(* IEC 61131-3 sources: cc_kush_rewrite/POUs (part 3) *)

FC_ModbusWriteBool(pRegisters := ADR(awModbusInputRegisters), iRegisterIndex := 355, iBitIndex := 0, xValue := stBunker[2].MotorVibrator[3].qxKM_Power);
FC_ModbusWriteBool(pRegisters := ADR(awModbusInputRegisters), iRegisterIndex := 355, iBitIndex := 1, xValue := stBunker[2].MotorVibrator[4].qxKM_Power);
FC_ModbusWriteBool(pRegisters := ADR(awModbusInputRegisters), iRegisterIndex := 355, iBitIndex := 2, xValue := stBunker[3].MotorVibFeeder[1].qxKM_Power);
FC_ModbusWriteBool(pRegisters := ADR(awModbusInputRegisters), iRegisterIndex := 355, iBitIndex := 3, xValue := stBunker[3].MotorVibFeeder[2].qxKM_Power);
FC_ModbusWriteBool(pRegisters := ADR(awModbusInputRegisters), iRegisterIndex := 355, iBitIndex := 4, xValue := stBunker[3].MotorVibrator[1].qxKM_Power);
FC_ModbusWriteBool(pRegisters := ADR(awModbusInputRegisters), iRegisterIndex := 355, iBitIndex := 5, xValue := stBunker[3].MotorVibrator[2].qxKM_Power);
FC_ModbusWriteBool(pRegisters := ADR(awModbusInputRegisters), iRegisterIndex := 355, iBitIndex := 6, xValue := stBunker[3].MotorVibrator[3].qxKM_Power);
FC_ModbusWriteBool(pRegisters := ADR(awModbusInputRegisters), iRegisterIndex := 355, iBitIndex := 7, xValue := stBunker[3].MotorVibrator[4].qxKM_Power);
FC_ModbusWriteBool(pRegisters := ADR(awModbusInputRegisters), iRegisterIndex := 355, iBitIndex := 8, xValue := stConveyor.xHLA);
FC_ModbusWriteBool(pRegisters := ADR(awModbusInputRegisters), iRegisterIndex := 355, iBitIndex := 10, xValue := stDumper.xHLA);
FC_ModbusWriteBool(pRegisters := ADR(awModbusInputRegisters), iRegisterIndex := 355, iBitIndex := 11, xValue := stCommonSignals.qx6KM1);
FC_ModbusWriteBool(pRegisters := ADR(awModbusInputRegisters), iRegisterIndex := 355, iBitIndex := 12, xValue := stConveyor.qxBreakerConveyor);
FC_ModbusWriteBool(pRegisters := ADR(awModbusInputRegisters), iRegisterIndex := 355, iBitIndex := 13, xValue := stDumper.qxBreakerConveyor);
FC_ModbusWriteBool(pRegisters := ADR(awModbusInputRegisters), iRegisterIndex := 355, iBitIndex := 14, xValue := stDumper.qxBreakerRotation);

// Модуль DO4 (356-357): Светофоры бункеров
FC_ModbusWriteBool(pRegisters := ADR(awModbusInputRegisters), iRegisterIndex := 356, iBitIndex := 0, xValue := stBunker[1].qxLightRed);
FC_ModbusWriteBool(pRegisters := ADR(awModbusInputRegisters), iRegisterIndex := 356, iBitIndex := 1, xValue := stBunker[1].qxLightYellow);
FC_ModbusWriteBool(pRegisters := ADR(awModbusInputRegisters), iRegisterIndex := 356, iBitIndex := 2, xValue := stBunker[1].qxLightGreen);
FC_ModbusWriteBool(pRegisters := ADR(awModbusInputRegisters), iRegisterIndex := 356, iBitIndex := 3, xValue := stBunker[2].qxLightRed);
FC_ModbusWriteBool(pRegisters := ADR(awModbusInputRegisters), iRegisterIndex := 356, iBitIndex := 4, xValue := stBunker[2].qxLightYellow);
FC_ModbusWriteBool(pRegisters := ADR(awModbusInputRegisters), iRegisterIndex := 356, iBitIndex := 5, xValue := stBunker[2].qxLightGreen);
FC_ModbusWriteBool(pRegisters := ADR(awModbusInputRegisters), iRegisterIndex := 356, iBitIndex := 6, xValue := stBunker[3].qxLightRed);
FC_ModbusWriteBool(pRegisters := ADR(awModbusInputRegisters), iRegisterIndex := 356, iBitIndex := 7, xValue := stBunker[3].qxLightYellow);
FC_ModbusWriteBool(pRegisters := ADR(awModbusInputRegisters), iRegisterIndex := 356, iBitIndex := 8, xValue := stBunker[3].qxLightGreen);

END_FUNCTION_BLOCK

(* ---- FB_Simulation.st ---- *)
FUNCTION_BLOCK FB_Simulation
VAR_INPUT
	xEnable : BOOL; // Включение симуляции
	xReset : BOOL; // Сброс всех переменных (симуляция отсутствия ошибок)
	Dumper : REFERENCE TO ST_Dumper; // Структура отвалообразователя
	Conveyor : REFERENCE TO ST_ConveyorPrefabricated; // Структура сборного конвейера
	Bunker : REFERENCE TO ARRAY[1..3] OF ST_Bunker; // Массив бункеров
	Common : ST_CommonSignals; // Общие сигналы
	tFeedbackDelay : TIME := T#500MS; // Задержка обратной связи
END_VAR
VAR
	// Детекция переднего фронта
	rtEnable : R_TRIG;
	rtReset : R_TRIG;

	// Флаг инициализации
	_xInitRequired : BOOL;

	// Индексы для циклов
	b, m : INT;

	// === Симуляция веса бункеров ===
	// Средняя частота вибропитателей каждого бункера
	_rAvgFrequencyVibFeeder : ARRAY[1..3] OF REAL;

	// Скорость расхода веса бункера (кг/с) в зависимости от частоты вибропитателей
	_rWeightDischargeRate : ARRAY[1..3] OF REAL;

	// Скорость заполнения веса бункера (кг/с) в зависимости от светофора
	_rWeightFillRate : ARRAY[1..3] OF REAL;

	// Таймер для периодического заполнения по приоритету
	_tonFillTimer : ARRAY[1..3] OF TON;
	_xFillTimerActive : ARRAY[1..3] OF BOOL;

	// Параметры заполнения (настраиваются через входные параметры)
	_rFillRateGreen : REAL := 0.8; // Скорость заполнения на зелёном (кг/с) - плавное заполнение
	_rFillRateYellow : REAL := 0.3; // Скорость заполнения на жёлтом (кг/с) - медленное заполнение
	_tFillPeriod : TIME := T#8S; // Период заполнения (раз в N секунд) - реже
	_tFillDuration : TIME := T#3S; // Длительность одного заполнения - дольше

	// Константа расхода: частота 50 Гц → 0.5 кг/с расход (замедлено)
	_rDischargeCoeff : REAL := 0.01; // 50 Гц * 0.01 = 0.5 кг/с

	// === Симуляция веса под бункерами ===

	// Скорость накопления веса (кг/с) для каждого бункера
	_rWeightAccumulationRate : ARRAY[1..3] OF REAL;

	// Накопленный вес от каждого бункера (независимо)
	_rLocalWeightUnderBunker : ARRAY[1..3] OF REAL;

	// === Случайные возмущения для бункеров ===
	// Параметры генератора псевдослучайных чисел (Linear Congruential Generator)
	_nRandomSeed : ARRAY[1..3] OF DINT := [12345, 67890, 24680]; // Начальные значения

	// Случайное смещение для каждого бункера (-1.0 до +1.0)
	_rRandomOffset : ARRAY[1..3] OF REAL;

	// Линейный дрейф (медленное изменение характеристик материала)
	_rDriftOffset : ARRAY[1..3] OF REAL;
	_rDriftSpeed : ARRAY[1..3] OF REAL := [0.0003, -0.00025, 0.00035]; // Скорость дрейфа за цикл

	// Временные переменные
	_rNoise : REAL; // Шум ±3%
	_rDrift : REAL; // Дрейф ±8%

	// === Таймеры отвалообразователя ===
	// Таймеры обратной связи контакторов (KM)
	tonKM_Conv1, tonKM_Conv2 : TON;
	tonKM_Rot1, tonKM_Rot2 : TON;

	// Таймеры обратной связи ЧРП (IsWorking)
	tonVFD_Conv1, tonVFD_Conv2 : TON;
	tonVFD_Rot1, tonVFD_Rot2 : TON;

	// Таймеры обратной связи тормозов отвалообразователя
	tonBreaker_DumperConv, tonBreaker_DumperRot : TON;

	// === Таймеры сборного конвейера ===
	// Таймеры обратной связи контакторов (KM)
	tonKM_PrefConv1, tonKM_PrefConv2 : TON;

	// Таймеры обратной связи ЧРП (IsWorking)
	tonVFD_PrefConv1, tonVFD_PrefConv2 : TON;

	// Таймер обратной связи тормоза сборного конвейера
	tonBreaker_PrefConv : TON;

	// === Таймеры бункеров ===
	// Таймеры обратной связи вибропитателей [бункер 1..3][мотор 1..2]
	tonKM_VibFeeder : ARRAY[1..3, 1..2] OF TON;
	tonVFD_VibFeeder : ARRAY[1..3, 1..2] OF TON;

	// Таймеры обратной связи вибраторов [бункер 1..3][мотор 1..4]
	tonKM_Vibrator : ARRAY[1..3, 1..4] OF TON;
	tonVFD_Vibrator : ARRAY[1..3, 1..4] OF TON;

	// ========================================
	// ПЕРЕМЕННЫЕ ДЛЯ ОТЛАДКИ - СИМУЛЯЦИЯ ОБРАТНОЙ СВЯЗИ VFD
	// TRUE = обратная связь есть (нормальная работа)
	// FALSE = обратная связь отсутствует (ошибка - нет обратной связи)
	// ========================================

	// Отвалообразователь - моторы конвейера
	_xSimVFDFeedback_DumperConv1 : BOOL := TRUE;
	_xSimVFDFeedback_DumperConv2 : BOOL := TRUE;

	// Отвалообразователь - моторы поворота
	_xSimVFDFeedback_DumperRot1 : BOOL := TRUE;
	_xSimVFDFeedback_DumperRot2 : BOOL := TRUE;

	// Сборный конвейер - моторы конвейера
	_xSimVFDFeedback_ConveyorConv1 : BOOL := TRUE;
	_xSimVFDFeedback_ConveyorConv2 : BOOL := TRUE;

	// Бункеры - вибропитатели [бункер 1..3][мотор 1..2]
	_xSimVFDFeedback_VibFeeder : ARRAY[1..3, 1..2] OF BOOL := [TRUE, TRUE, TRUE, TRUE, TRUE, TRUE];

	// Бункеры - вибраторы [бункер 1..3][мотор 1..4]
	_xSimVFDFeedback_Vibrator : ARRAY[1..3, 1..4] OF BOOL := [
		TRUE, TRUE, TRUE, TRUE,
		TRUE, TRUE, TRUE, TRUE,
		TRUE, TRUE, TRUE, TRUE
	];
END_VAR

// Детекция фронтов
rtEnable(CLK := xEnable);
rtReset(CLK := xReset);

// Инициализация по переднему фронту Enable или Reset
_xInitRequired := rtEnable.Q OR rtReset.Q;

IF _xInitRequired THEN

	// ========================================
	// ИНИЦИАЛИЗАЦИЯ ОБЩИЕ СИГНАЛЫ
	// ========================================

	// Кнопка аварийной остановки - инвертированный сигнал (NC)
	Common.fbEmergencyStopBtn.ixSignal := TRUE;

	// Сигнал ПМУ - режим управления 1 - дистанция, 0 - местный
	Common.fbRemoteModeBtn.ixSignal := TRUE;

	// ========================================
	// ИНИЦИАЛИЗАЦИЯ СИМУЛЯЦИИ ОТВАЛООБРАЗОВАТЕЛЯ
	// Установка всех сигналов в состояние "нет ошибок"
	// ========================================

	// Моторы конвейера - ЧРП готовность
	Dumper.MotorConveyor[1].VFD.fbStateRdyToStart.ixSignal := TRUE;
	Dumper.MotorConveyor[2].VFD.fbStateRdyToStart.ixSignal := TRUE;

	// Моторы поворота - ЧРП готовность
	Dumper.MotorRotation[1].VFD.fbStateRdyToStart.ixSignal := TRUE;
	Dumper.MotorRotation[2].VFD.fbStateRdyToStart.ixSignal := TRUE;

	// Автоматические выключатели (QF)
	Dumper.MotorConveyor[1].fbStateQF.ixSignal := TRUE;
	Dumper.MotorConveyor[2].fbStateQF.ixSignal := TRUE;
	Dumper.MotorRotation[1].fbStateQF.ixSignal := TRUE;
	Dumper.MotorRotation[2].fbStateQF.ixSignal := TRUE;

	// ЧРП ошибки - инвертированный сигнал (NC)
	Dumper.MotorConveyor[1].VFD.fbStateFailure.ixSignal := TRUE;
	Dumper.MotorConveyor[2].VFD.fbStateFailure.ixSignal := TRUE;
	Dumper.MotorRotation[1].VFD.fbStateFailure.ixSignal := TRUE;
	Dumper.MotorRotation[2].VFD.fbStateFailure.ixSignal := TRUE;

	// Перегрев статора - инвертированный сигнал (NC)
	Dumper.MotorConveyor[1].fbStatorOverheat.ixSignal := TRUE;
	Dumper.MotorConveyor[2].fbStatorOverheat.ixSignal := TRUE;
	Dumper.MotorRotation[1].fbStatorOverheat.ixSignal := TRUE;
	Dumper.MotorRotation[2].fbStatorOverheat.ixSignal := TRUE;

	// Кабель-тросовые выключатели (HQ)
	Dumper.fbHQ_IsOk[1].ixSignal := TRUE;
	Dumper.fbHQ_IsOk[2].ixSignal := TRUE;
	Dumper.fbHQ_IsOk[3].ixSignal := TRUE;
	Dumper.fbHQ_IsOk[4].ixSignal := TRUE;

	// Контроль ограждения барабана (SQ)
	Dumper.fbSQ_IsOk[1].ixSignal := TRUE;
	Dumper.fbSQ_IsOk[2].ixSignal := TRUE;

	// Контроль схода ленты - тревога (ZQ) - инвертированный сигнал (NC)
	Dumper.fbZQAlarm[1].ixSignal := TRUE;
	Dumper.fbZQAlarm[2].ixSignal := TRUE;
	Dumper.fbZQAlarm[3].ixSignal := TRUE;
	Dumper.fbZQAlarm[4].ixSignal := TRUE;

	// Контроль схода ленты - предупреждение (ZQ) - инвертированный сигнал (NC)
	Dumper.fbZQWarning[1].ixSignal := TRUE;
	Dumper.fbZQWarning[2].ixSignal := TRUE;
	Dumper.fbZQWarning[3].ixSignal := TRUE;
	Dumper.fbZQWarning[4].ixSignal := TRUE;

	// Кнопка аварийной остановки - инвертированный сигнал (NC)
	Dumper.fbBtnEmergencyStop.ixSignal := TRUE;

	// Концевые выключатели - инвертированный сигнал (NC)
	Dumper.fbEndSwitchLeft.ixSignal := TRUE;
	Dumper.fbEndSwitchRight.ixSignal := TRUE;

	// Контроль заштыбовки - норма = 1
	Dumper.fbGS1.ixSignal := TRUE;

	// Контроль продольного разрыва ленты - норма = 1
	Dumper.fbYS1.ixSignal := TRUE;

	// Тормоза - в начале активны (NOT released)
	Dumper.fbBreakerConveyor.ixSignal := FALSE;
	Dumper.fbBreakerRotation.ixSignal := FALSE;

	// ========================================
	// ИНИЦИАЛИЗАЦИЯ СИМУЛЯЦИИ СБОРНОГО КОНВЕЙЕРА
	// Установка всех сигналов в состояние "нет ошибок"
	// ========================================

	// Моторы конвейера - ЧРП готовность
	Conveyor.MotorConveyor[1].VFD.fbStateRdyToStart.ixSignal := TRUE;
	Conveyor.MotorConveyor[2].VFD.fbStateRdyToStart.ixSignal := TRUE;

	// Автоматические выключатели (QF)
	Conveyor.MotorConveyor[1].fbStateQF.ixSignal := TRUE;
	Conveyor.MotorConveyor[2].fbStateQF.ixSignal := TRUE;

	// ЧРП ошибки - инвертированный сигнал (NC)
	Conveyor.MotorConveyor[1].VFD.fbStateFailure.ixSignal := TRUE;
	Conveyor.MotorConveyor[2].VFD.fbStateFailure.ixSignal := TRUE;

	// Перегрев статора - инвертированный сигнал (NC)
	Conveyor.MotorConveyor[1].fbStatorOverheat.ixSignal := TRUE;
	Conveyor.MotorConveyor[2].fbStatorOverheat.ixSignal := TRUE;

	// Кабель-тросовые выключатели (HQ)
	Conveyor.fbHQ_IsOk[1].ixSignal := TRUE;
	Conveyor.fbHQ_IsOk[2].ixSignal := TRUE;
	Conveyor.fbHQ_IsOk[3].ixSignal := TRUE;
	Conveyor.fbHQ_IsOk[4].ixSignal := TRUE;

	// Контроль ограждения барабана (SQ)
	Conveyor.fbSQ_IsOk[1].ixSignal := TRUE;
	Conveyor.fbSQ_IsOk[2].ixSignal := TRUE;

	// Контроль схода ленты - тревога (ZQ) - инвертированный сигнал (NC)
	Conveyor.fbZQAlarm[1].ixSignal := TRUE;
	Conveyor.fbZQAlarm[2].ixSignal := TRUE;
	Conveyor.fbZQAlarm[3].ixSignal := TRUE;
	Conveyor.fbZQAlarm[4].ixSignal := TRUE;

	// Контроль схода ленты - предупреждение (ZQ) - инвертированный сигнал (NC)
	Conveyor.fbZQWarning[1].ixSignal := TRUE;
	Conveyor.fbZQWarning[2].ixSignal := TRUE;
	Conveyor.fbZQWarning[3].ixSignal := TRUE;
	Conveyor.fbZQWarning[4].ixSignal := TRUE;

	// Кнопка аварийной остановки - инвертированный сигнал (NC)
	Conveyor.fbBtnEmergencyStop.ixSignal := TRUE;

	// Контроль заштыбовки - норма = 1
	Conveyor.fbGS1.ixSignal := TRUE;

	// Контроль продольного разрыва ленты - норма = 1
	Conveyor.fbYS1.ixSignal := TRUE;

	// Металлодетектор - норма = 0 (металл не обнаружен)
	Conveyor.fbYE1.ixSignal := FALSE;

	// ========================================
	// ИНИЦИАЛИЗАЦИЯ СИМУЛЯЦИИ БУНКЕРОВ
	// Установка всех сигналов в состояние "нет ошибок"
	// ========================================

	// ========================================
	// БУНКЕР 1
	// ========================================

	// Вибропитатели (MotorVibFeeder[1..2])
	// Вибропитатель 1
	Bunker[1].MotorVibFeeder[1].VFD.fbStateRdyToStart.ixSignal := TRUE;
	Bunker[1].MotorVibFeeder[1].fbStateQF.ixSignal := TRUE;
	Bunker[1].MotorVibFeeder[1].VFD.fbStateFailure.ixSignal := TRUE;
	Bunker[1].MotorVibFeeder[1].fbStatorOverheat.ixSignal := TRUE;

	// Вибропитатель 2
	Bunker[1].MotorVibFeeder[2].VFD.fbStateRdyToStart.ixSignal := TRUE;
	Bunker[1].MotorVibFeeder[2].fbStateQF.ixSignal := TRUE;
	Bunker[1].MotorVibFeeder[2].VFD.fbStateFailure.ixSignal := TRUE;
	Bunker[1].MotorVibFeeder[2].fbStatorOverheat.ixSignal := TRUE;

	// Вибраторы (MotorVibrator[1..4])
	Bunker[1].MotorVibrator[1].VFD.fbStateRdyToStart.ixSignal := TRUE;
	Bunker[1].MotorVibrator[1].fbStateQF.ixSignal := TRUE;
	Bunker[1].MotorVibrator[1].VFD.fbStateFailure.ixSignal := TRUE;

	Bunker[1].MotorVibrator[2].VFD.fbStateRdyToStart.ixSignal := TRUE;
	Bunker[1].MotorVibrator[2].fbStateQF.ixSignal := TRUE;
	Bunker[1].MotorVibrator[2].VFD.fbStateFailure.ixSignal := TRUE;

	Bunker[1].MotorVibrator[3].VFD.fbStateRdyToStart.ixSignal := TRUE;
	Bunker[1].MotorVibrator[3].fbStateQF.ixSignal := TRUE;
	Bunker[1].MotorVibrator[3].VFD.fbStateFailure.ixSignal := TRUE;

	Bunker[1].MotorVibrator[4].VFD.fbStateRdyToStart.ixSignal := TRUE;
	Bunker[1].MotorVibrator[4].fbStateQF.ixSignal := TRUE;
	Bunker[1].MotorVibrator[4].VFD.fbStateFailure.ixSignal := TRUE;

	// Люк бункера - закрыт (норма = 1)
	Bunker[1].fbStateHatch.ixSignal := TRUE;

	// Кнопка аварийной остановки - инвертированный сигнал (NC)
	Bunker[1].fbBtnEmergencyStop.ixSignal := TRUE;

	// Начальный вес бункера (симуляция заполненного бункера)
	Bunker[1].rWeight := 100.0;

	// Сброс веса под бункером
	Bunker[1].rWeightUnderBunker := 0.0;
	_rLocalWeightUnderBunker[1] := 0.0;

	// Сброс дрейфа
	_rDriftOffset[1] := 0.0;

	// ========================================
	// БУНКЕР 2
	// ========================================

	// Вибропитатели (MotorVibFeeder[1..2])
	// Вибропитатель 1
	Bunker[2].MotorVibFeeder[1].VFD.fbStateRdyToStart.ixSignal := TRUE;
	Bunker[2].MotorVibFeeder[1].fbStateQF.ixSignal := TRUE;
	Bunker[2].MotorVibFeeder[1].VFD.fbStateFailure.ixSignal := TRUE;
	Bunker[2].MotorVibFeeder[1].fbStatorOverheat.ixSignal := TRUE;

	// Вибропитатель 2
	Bunker[2].MotorVibFeeder[2].VFD.fbStateRdyToStart.ixSignal := TRUE;
	Bunker[2].MotorVibFeeder[2].fbStateQF.ixSignal := TRUE;
	Bunker[2].MotorVibFeeder[2].VFD.fbStateFailure.ixSignal := TRUE;
	Bunker[2].MotorVibFeeder[2].fbStatorOverheat.ixSignal := TRUE;

	// Вибраторы (MotorVibrator[1..4])
	Bunker[2].MotorVibrator[1].VFD.fbStateRdyToStart.ixSignal := TRUE;
	Bunker[2].MotorVibrator[1].fbStateQF.ixSignal := TRUE;
	Bunker[2].MotorVibrator[1].VFD.fbStateFailure.ixSignal := TRUE;

	Bunker[2].MotorVibrator[2].VFD.fbStateRdyToStart.ixSignal := TRUE;
	Bunker[2].MotorVibrator[2].fbStateQF.ixSignal := TRUE;
	Bunker[2].MotorVibrator[2].VFD.fbStateFailure.ixSignal := TRUE;

	Bunker[2].MotorVibrator[3].VFD.fbStateRdyToStart.ixSignal := TRUE;
	Bunker[2].MotorVibrator[3].fbStateQF.ixSignal := TRUE;
	Bunker[2].MotorVibrator[3].VFD.fbStateFailure.ixSignal := TRUE;

	Bunker[2].MotorVibrator[4].VFD.fbStateRdyToStart.ixSignal := TRUE;
	Bunker[2].MotorVibrator[4].fbStateQF.ixSignal := TRUE;
	Bunker[2].MotorVibrator[4].VFD.fbStateFailure.ixSignal := TRUE;

	// Люк бункера - закрыт (норма = 1)
	Bunker[2].fbStateHatch.ixSignal := TRUE;

	// Кнопка аварийной остановки - инвертированный сигнал (NC)
	Bunker[2].fbBtnEmergencyStop.ixSignal := TRUE;

	// Начальный вес бункера (симуляция заполненного бункера)
	Bunker[2].rWeight := 100.0;

	// Сброс веса под бункером
	Bunker[2].rWeightUnderBunker := 0.0;
	_rLocalWeightUnderBunker[2] := 0.0;

	// Сброс дрейфа
	_rDriftOffset[2] := 0.0;

	// ========================================
	// БУНКЕР 3
	// ========================================

	// Вибропитатели (MotorVibFeeder[1..2])
	// Вибропитатель 1
	Bunker[3].MotorVibFeeder[1].VFD.fbStateRdyToStart.ixSignal := TRUE;
	Bunker[3].MotorVibFeeder[1].fbStateQF.ixSignal := TRUE;
	Bunker[3].MotorVibFeeder[1].VFD.fbStateFailure.ixSignal := TRUE;
	Bunker[3].MotorVibFeeder[1].fbStatorOverheat.ixSignal := TRUE;

	// Вибропитатель 2
	Bunker[3].MotorVibFeeder[2].VFD.fbStateRdyToStart.ixSignal := TRUE;
	Bunker[3].MotorVibFeeder[2].fbStateQF.ixSignal := TRUE;
	Bunker[3].MotorVibFeeder[2].VFD.fbStateFailure.ixSignal := TRUE;
	Bunker[3].MotorVibFeeder[2].fbStatorOverheat.ixSignal := TRUE;

	// Вибраторы (MotorVibrator[1..4])
	Bunker[3].MotorVibrator[1].VFD.fbStateRdyToStart.ixSignal := TRUE;
	Bunker[3].MotorVibrator[1].fbStateQF.ixSignal := TRUE;
	Bunker[3].MotorVibrator[1].VFD.fbStateFailure.ixSignal := TRUE;

	Bunker[3].MotorVibrator[2].VFD.fbStateRdyToStart.ixSignal := TRUE;
	Bunker[3].MotorVibrator[2].fbStateQF.ixSignal := TRUE;
	Bunker[3].MotorVibrator[2].VFD.fbStateFailure.ixSignal := TRUE;

	Bunker[3].MotorVibrator[3].VFD.fbStateRdyToStart.ixSignal := TRUE;
	Bunker[3].MotorVibrator[3].fbStateQF.ixSignal := TRUE;
	Bunker[3].MotorVibrator[3].VFD.fbStateFailure.ixSignal := TRUE;

	Bunker[3].MotorVibrator[4].VFD.fbStateRdyToStart.ixSignal := TRUE;
	Bunker[3].MotorVibrator[4].fbStateQF.ixSignal := TRUE;
	Bunker[3].MotorVibrator[4].VFD.fbStateFailure.ixSignal := TRUE;

	// Люк бункера - закрыт (норма = 1)
	Bunker[3].fbStateHatch.ixSignal := TRUE;

	// Кнопка аварийной остановки - инвертированный сигнал (NC)
	Bunker[3].fbBtnEmergencyStop.ixSignal := TRUE;

	// Начальный вес бункера (симуляция заполненного бункера)
	Bunker[3].rWeight := 100.0;

	// Сброс веса под бункером
	Bunker[3].rWeightUnderBunker := 0.0;
	_rLocalWeightUnderBunker[3] := 0.0;

	// Сброс дрейфа
	_rDriftOffset[3] := 0.0;
END_IF;

// ========================================
// ПРОЦЕСС СИМУЛЯЦИИ
// ========================================

IF xEnable THEN
	// ========================================
	// СИМУЛЯЦИЯ ОТВАЛООБРАЗОВАТЕЛЯ
	// ========================================

	// Симуляция частоты ЧРП моторов конвейера отвалообразователя
	// В режиме симуляции FB_AnalogInput использует refSimValue (rSimulatedFrequency) напрямую,
	// поэтому записываем целевую частоту в rSimulatedFrequency
	Dumper.MotorConveyor[1].VFD.rSimulatedFrequency := Dumper.MotorConveyor[1].VFD.qrOutFrequency;
	Dumper.MotorConveyor[2].VFD.rSimulatedFrequency := Dumper.MotorConveyor[2].VFD.qrOutFrequency;

	// Симуляция частоты ЧРП моторов поворота отвалообразователя
	Dumper.MotorRotation[1].VFD.rSimulatedFrequency := Dumper.MotorRotation[1].VFD.qrOutFrequency;
	Dumper.MotorRotation[2].VFD.rSimulatedFrequency := Dumper.MotorRotation[2].VFD.qrOutFrequency;

	// ========================================
	// СИМУЛЯЦИЯ ОБРАТНОЙ СВЯЗИ ОТВАЛООБРАЗОВАТЕЛЯ
	// ========================================

	// Обратная связь контакторов моторов конвейера отвалообразователя
	tonKM_Conv1(IN := Dumper.MotorConveyor[1].qxKM_Power, PT := tFeedbackDelay);
	Dumper.MotorConveyor[1].fbStateKM.ixSignal := tonKM_Conv1.Q;

	tonKM_Conv2(IN := Dumper.MotorConveyor[2].qxKM_Power, PT := tFeedbackDelay);
	Dumper.MotorConveyor[2].fbStateKM.ixSignal := tonKM_Conv2.Q;

	// Обратная связь контакторов моторов поворота отвалообразователя
	tonKM_Rot1(IN := Dumper.MotorRotation[1].qxKM_Power, PT := tFeedbackDelay);
	Dumper.MotorRotation[1].fbStateKM.ixSignal := tonKM_Rot1.Q;

	tonKM_Rot2(IN := Dumper.MotorRotation[2].qxKM_Power, PT := tFeedbackDelay);
	Dumper.MotorRotation[2].fbStateKM.ixSignal := tonKM_Rot2.Q;

	// Обратная связь работы ЧРП моторов конвейера отвалообразователя
	tonVFD_Conv1(IN := Dumper.MotorConveyor[1].VFD.qxStart, PT := tFeedbackDelay);
	Dumper.MotorConveyor[1].VFD.fbStateIsWorking.ixSignal := tonVFD_Conv1.Q AND _xSimVFDFeedback_DumperConv1;

	tonVFD_Conv2(IN := Dumper.MotorConveyor[2].VFD.qxStart, PT := tFeedbackDelay);
	Dumper.MotorConveyor[2].VFD.fbStateIsWorking.ixSignal := tonVFD_Conv2.Q AND _xSimVFDFeedback_DumperConv2;

	// Обратная связь работы ЧРП моторов поворота отвалообразователя
	// Учитываем как прямое, так и реверсивное вращение
	tonVFD_Rot1(IN := (Dumper.MotorRotation[1].VFD.qxStart OR Dumper.MotorRotation[1].qxVFDReverseStart), PT := tFeedbackDelay);
	Dumper.MotorRotation[1].VFD.fbStateIsWorking.ixSignal := tonVFD_Rot1.Q AND _xSimVFDFeedback_DumperRot1;

	tonVFD_Rot2(IN := (Dumper.MotorRotation[2].VFD.qxStart OR Dumper.MotorRotation[2].qxVFDReverseStart), PT := tFeedbackDelay);
	Dumper.MotorRotation[2].VFD.fbStateIsWorking.ixSignal := tonVFD_Rot2.Q AND _xSimVFDFeedback_DumperRot2;

	// Обратная связь тормозов отвалообразователя
	// Тормоз отпущен (TRUE) когда на выходе активен сигнал
	// Тормоз активен (FALSE) когда выход отключен
	tonBreaker_DumperConv(IN := Dumper.qxBreakerConveyor, PT := tFeedbackDelay);
	Dumper.fbBreakerConveyor.ixSignal := tonBreaker_DumperConv.Q;

	tonBreaker_DumperRot(IN := Dumper.qxBreakerRotation, PT := tFeedbackDelay);
	Dumper.fbBreakerRotation.ixSignal := tonBreaker_DumperRot.Q;

	// ========================================
	// СИМУЛЯЦИЯ СБОРНОГО КОНВЕЙЕРА
	// ========================================

	// Симуляция частоты ЧРП моторов конвейера
	// В режиме симуляции FB_AnalogInput использует refSimValue (rSimulatedFrequency) напрямую,
	// поэтому записываем целевую частоту в rSimulatedFrequency
	Conveyor.MotorConveyor[1].VFD.rSimulatedFrequency := Conveyor.MotorConveyor[1].VFD.qrOutFrequency;
	Conveyor.MotorConveyor[2].VFD.rSimulatedFrequency := Conveyor.MotorConveyor[2].VFD.qrOutFrequency;

	// ========================================
	// СИМУЛЯЦИЯ ОБРАТНОЙ СВЯЗИ СБОРНОГО КОНВЕЙЕРА
	// ========================================

	// Обратная связь контакторов моторов конвейера
	tonKM_PrefConv1(IN := Conveyor.MotorConveyor[1].qxKM_Power, PT := tFeedbackDelay);
	Conveyor.MotorConveyor[1].fbStateKM.ixSignal := tonKM_PrefConv1.Q;

	tonKM_PrefConv2(IN := Conveyor.MotorConveyor[2].qxKM_Power, PT := tFeedbackDelay);
	Conveyor.MotorConveyor[2].fbStateKM.ixSignal := tonKM_PrefConv2.Q;

	// Обратная связь работы ЧРП моторов конвейера
	tonVFD_PrefConv1(IN := Conveyor.MotorConveyor[1].VFD.qxStart, PT := tFeedbackDelay);
	Conveyor.MotorConveyor[1].VFD.fbStateIsWorking.ixSignal := tonVFD_PrefConv1.Q AND _xSimVFDFeedback_ConveyorConv1;

	tonVFD_PrefConv2(IN := Conveyor.MotorConveyor[2].VFD.qxStart, PT := tFeedbackDelay);
	Conveyor.MotorConveyor[2].VFD.fbStateIsWorking.ixSignal := tonVFD_PrefConv2.Q AND _xSimVFDFeedback_ConveyorConv2;

	// Обратная связь тормоза сборного конвейера
	tonBreaker_PrefConv(IN := Conveyor.qxBreakerConveyor, PT := tFeedbackDelay);
	Conveyor.fbBreakerConveyor.ixSignal := tonBreaker_PrefConv.Q;

	// ========================================
	// СИМУЛЯЦИЯ БУНКЕРОВ
	// ========================================

	FOR b := 1 TO 3 BY 1 DO
		// --- Вибропитатели (MotorVibFeeder[1..2]) ---
		FOR m := 1 TO 2 BY 1 DO
			// Симуляция частоты ЧРП вибропитателя
			// В режиме симуляции FB_AnalogInput использует refSimValue (rSimulatedFrequency) напрямую,
			// поэтому записываем целевую частоту в rSimulatedFrequency
			Bunker[b].MotorVibFeeder[m].VFD.rSimulatedFrequency := Bunker[b].MotorVibFeeder[m].VFD.qrOutFrequency;

			// Обратная связь контактора вибропитателя
			tonKM_VibFeeder[b, m](IN := Bunker[b].MotorVibFeeder[m].qxKM_Power, PT := tFeedbackDelay);
			Bunker[b].MotorVibFeeder[m].fbStateKM.ixSignal := tonKM_VibFeeder[b, m].Q;

			// Обратная связь работы ЧРП вибропитателя
			tonVFD_VibFeeder[b, m](IN := Bunker[b].MotorVibFeeder[m].VFD.qxStart, PT := tFeedbackDelay);
			Bunker[b].MotorVibFeeder[m].VFD.fbStateIsWorking.ixSignal := tonVFD_VibFeeder[b, m].Q AND _xSimVFDFeedback_VibFeeder[b, m];
		END_FOR;

		// --- Вибраторы (MotorVibrator[1..4]) ---
		FOR m := 1 TO 4 BY 1 DO
			// Симуляция частоты ЧРП вибратора
			// В режиме симуляции FB_AnalogInput использует refSimValue (rSimulatedFrequency) напрямую,
			// поэтому записываем целевую частоту в rSimulatedFrequency
			Bunker[b].MotorVibrator[m].VFD.rSimulatedFrequency := Bunker[b].MotorVibrator[m].VFD.qrOutFrequency;

			// Обратная связь контактора вибратора
			tonKM_Vibrator[b, m](IN := Bunker[b].MotorVibrator[m].qxKM_Power, PT := tFeedbackDelay);
			Bunker[b].MotorVibrator[m].fbStateKM.ixSignal := tonKM_Vibrator[b, m].Q;

			// Обратная связь работы ЧРП вибратора
			tonVFD_Vibrator[b, m](IN := Bunker[b].MotorVibrator[m].VFD.qxStart, PT := tFeedbackDelay);
			Bunker[b].MotorVibrator[m].VFD.fbStateIsWorking.ixSignal := tonVFD_Vibrator[b, m].Q AND _xSimVFDFeedback_Vibrator[b, m];
		END_FOR;
	END_FOR;

	// ========================================
	// СИМУЛЯЦИЯ ВЕСА ПОД БУНКЕРАМИ
	// ========================================

	// Симуляция с случайными возмущениями для тестирования ПИД-регулятора
	FOR b := 1 TO 3 BY 1 DO
		// Средняя выходная частота двух вибропитателей бункера
		// Используем rActualFrequency - актуальная частота от модуля AI (после полного цикла AO → AI)
		_rAvgFrequencyVibFeeder[b] :=
			(Bunker[b].MotorVibFeeder[1].VFD.rActualFrequency
		   + Bunker[b].MotorVibFeeder[2].VFD.rActualFrequency) / 2.0;

		// --- Генерация случайного шума (Linear Congruential Generator) ---
		// LCG формула: seed = (a * seed + c) mod m
		// Параметры: a = 1103515245, c = 12345, m = 2^31
		_nRandomSeed[b] := (1103515245 * _nRandomSeed[b] + 12345) MOD 2147483647;

		// Преобразование seed в диапазон [-1.0 ... +1.0]
		_rRandomOffset[b] := (DINT_TO_REAL(_nRandomSeed[b]) / 2147483647.0) * 2.0 - 1.0;

		// Шум ±3% от базового значения
		_rNoise := _rRandomOffset[b] * 0.03;

		// --- Медленный линейный дрейф (имитация изменения свойств материала) ---
		// Дрейф накапливается с течением времени, но ограничен диапазоном ±8%
		_rDriftOffset[b] := _rDriftOffset[b] + _rDriftSpeed[b];

		// Ограничение дрейфа в диапазоне [-0.08 ... +0.08]
		IF _rDriftOffset[b] > 0.08 THEN
			_rDriftOffset[b] := 0.08;
			_rDriftSpeed[b] := -ABS(_rDriftSpeed[b]); // Реверс направления
		ELSIF _rDriftOffset[b] < -0.08 THEN
			_rDriftOffset[b] := -0.08;
			_rDriftSpeed[b] := ABS(_rDriftSpeed[b]); // Реверс направления
		END_IF;

		_rDrift := _rDriftOffset[b];

		// --- Расчет веса с возмущениями ---
		// Базовая линейная зависимость: частота 50 Гц -> 100 кг
		// + Шум ±3%
		// + Дрейф ±8%
		_rLocalWeightUnderBunker[b] := (_rAvgFrequencyVibFeeder[b] / 50.0) * 100.0
		                             * (1.0 + _rNoise + _rDrift);

		// Ограничение минимального значения (вес не может быть отрицательным)
		IF _rLocalWeightUnderBunker[b] < 0.0 THEN
			_rLocalWeightUnderBunker[b] := 0.0;
		END_IF;
	END_FOR;

	// --- Формирование кумулятивных весов согласно движению конвейера ---
	// Конвейер движется: Бункер 3 → Бункер 2 → Бункер 1 → дальше
	//
	// rWeightUnderBunker[3] = вес только от бункера 3
	// rWeightUnderBunker[2] = вес от бункера 3 + вес от бункера 2
	// rWeightUnderBunker[1] = вес от бункера 3 + вес от бункера 2 + вес от бункера 1

	Bunker[3].rWeightUnderBunker := _rLocalWeightUnderBunker[3];

	Bunker[2].rWeightUnderBunker := _rLocalWeightUnderBunker[3]
	                              + _rLocalWeightUnderBunker[2];

	Bunker[1].rWeightUnderBunker := _rLocalWeightUnderBunker[3]
	                              + _rLocalWeightUnderBunker[2]
	                              + _rLocalWeightUnderBunker[1];

	// ========================================
	// СИМУЛЯЦИЯ ВЕСА БУНКЕРОВ (РАСХОД И ЗАПОЛНЕНИЕ)
	// ========================================

	IF SIMULATION_BUNKER_WEIGHT THEN
		FOR b := 1 TO 3 BY 1 DO
		// ========================================
		// 1. РАСХОД ВЕСА (пропорционален частоте вибропитателей)
		// ========================================

		// Средняя частота вибропитателей
		_rAvgFrequencyVibFeeder[b] :=
			(Bunker[b].MotorVibFeeder[1].VFD.rActualFrequency
		   + Bunker[b].MotorVibFeeder[2].VFD.rActualFrequency) / 2.0;

		// Скорость расхода (кг/с): частота * коэффициент
		// Пример: 50 Гц * 0.02 = 1.0 кг/с
		_rWeightDischargeRate[b] := _rAvgFrequencyVibFeeder[b] * _rDischargeCoeff;

		// Применение расхода к весу бункера (за один цикл ПЛК ~10-50 мс)
		// Предполагаем цикл ПЛК = 50 мс = 0.05 с
		Bunker[b].rWeight := Bunker[b].rWeight - (_rWeightDischargeRate[b] * 0.05);

		// Ограничение минимального веса (не может быть отрицательным)
		IF Bunker[b].rWeight < 0.0 THEN
			Bunker[b].rWeight := 0.0;
		END_IF;

		// ========================================
		// 2. ЗАПОЛНЕНИЕ ВЕСА (зависит от цвета светофора)
		// ========================================

		// Определение скорости заполнения в зависимости от цвета светофора
		CASE Bunker[b].eLightColor OF
			E_LightColor.GREEN:
				// Зелёный - максимальная скорость заполнения (приоритет)
				_rWeightFillRate[b] := _rFillRateGreen;

			E_LightColor.YELLOW:
				// Жёлтый - умеренная скорость заполнения
				_rWeightFillRate[b] := _rFillRateYellow;

			E_LightColor.RED, E_LightColor.OFF:
				// Красный или выключен - заполнение отсутствует
				_rWeightFillRate[b] := 0.0;
		END_CASE;

		// ========================================
		// 3. ПЕРИОДИЧЕСКОЕ ЗАПОЛНЕНИЕ (раз в N секунд)
		// ========================================

		// Таймер периода ожидания между заполнениями
		_tonFillTimer[b](
			IN := NOT _xFillTimerActive[b] AND (_rWeightFillRate[b] > 0.0),
			PT := _tFillPeriod
		);

		// Когда таймер ожидания истёк - запускаем процесс заполнения
		IF _tonFillTimer[b].Q THEN
			_xFillTimerActive[b] := TRUE;
			_tonFillTimer[b].IN := FALSE; // Сброс таймера ожидания
		END_IF;

		// Таймер длительности заполнения
		IF _xFillTimerActive[b] THEN
			// Применение заполнения к весу бункера (за один цикл ПЛК)
			Bunker[b].rWeight := Bunker[b].rWeight + (_rWeightFillRate[b] * 0.05);

			// Ограничение максимального веса (100 кг = 100%)
			IF Bunker[b].rWeight > 100.0 THEN
				Bunker[b].rWeight := 100.0;
			END_IF;

			// Проверка длительности заполнения
			_tonFillTimer[b](IN := TRUE, PT := _tFillDuration);

			// Когда заполнение завершено - сбросить флаг
			IF _tonFillTimer[b].Q THEN
				_xFillTimerActive[b] := FALSE;
				_tonFillTimer[b].IN := FALSE; // Сброс таймера заполнения
			END_IF;
		END_IF;

		// ========================================
		// 4. ПРИОРИТЕТ ЗЕЛЁНОГО СВЕТОФОРА
		// ========================================
		// Если хотя бы один бункер горит зелёным (критический режим),
		// то только он получает заполнение, а остальные ждут

		// Проверка: есть ли бункеры с зелёным светофором в критическом режиме?
		// (вес <= BUNKER_WEIGHT_LIGHT_RED_SPECIAL)
		IF (Bunker[1].eLightColor = E_LightColor.GREEN AND Bunker[1].rWeight <= BUNKER_WEIGHT_LIGHT_RED_SPECIAL)
		OR (Bunker[2].eLightColor = E_LightColor.GREEN AND Bunker[2].rWeight <= BUNKER_WEIGHT_LIGHT_RED_SPECIAL)
		OR (Bunker[3].eLightColor = E_LightColor.GREEN AND Bunker[3].rWeight <= BUNKER_WEIGHT_LIGHT_RED_SPECIAL)
		THEN
			// Есть критический бункер с зелёным светофором
			// Отменяем заполнение для всех НЕ критических бункеров
			IF Bunker[b].eLightColor <> E_LightColor.GREEN OR Bunker[b].rWeight > BUNKER_WEIGHT_LIGHT_RED_SPECIAL THEN
				_rWeightFillRate[b] := 0.0;
				_xFillTimerActive[b] := FALSE;
			END_IF;
		END_IF;
		END_FOR;
	END_IF; // IF SIMULATION_BUNKER_WEIGHT THEN

END_IF; // IF _xInitRequired THEN

END_FUNCTION_BLOCK

(* ---- MAIN.st ---- *)
PROGRAM MAIN
VAR
	fbSimulation : FB_Simulation;
	fbEmergencyStopCollector : FB_EmergencyStopCollector; // Централизованный сбор сигналов аварийной остановки
	fbScadaCommunication : FB_ScadaCommunication;
	fbModbusToSCADA : FB_ModbusToSCADA;

	fbBunker : ARRAY [1..3] OF FB_BunkerControl;
	stBunker : ARRAY [1..3] OF ST_Bunker;

	fbDumper : FB_DumperControl;
	stDumper : ST_Dumper;
	xStartDumper : BOOL := FALSE; // Команда запуска отвалообразователя
	xManualStopDumper : BOOL; // Ручная остановка отвалообразователя
	eDumperStage : E_StageWithPreStartAlarm; // Стадия отвалообразователя
	eDumperStageToSCADA : E_ScadaStatesDevice; // Состояние для SCADA отвалообразователя

	fbProportionPid : FB_ProportionPID;
	tonPidTimer : TON; // Таймер для периодического вызова ПИД
	xPidTimerPulse : BOOL := FALSE; // Импульс для вызова ПИД
	rtPidPulse : R_TRIG; // Детектор переднего фронта импульса

	fbConveyor : FB_ConveyorControl;
	stConveyor : ST_ConveyorPrefabricated;
	xStartConveyor : BOOL := FALSE; // Команда запуска конвейера
	xManualStopConveyor : BOOL; // Команда остановки сборного конвейера
	eConveyorStage : E_StageWithPreStartAlarm; // Стадия конвейера
	eConveyorStageToSCADA : E_ScadaStatesDevice; // Состояние для SCADA конвейера

	xStartBunker : ARRAY[1..3] OF BOOL := [FALSE, FALSE, FALSE]; // Команды запуска бункеров
	xManualStopBunker : ARRAY[1..3] OF BOOL; // Команды остановки бункеров
	eBunkerStage : ARRAY[1..3] OF E_StageWithPreStartAlarm; // Стадии бункеров
	eBunkerStageToSCADA : ARRAY[1..3] OF E_ScadaStatesDevice; // Состояния для SCADA бункеров

	stCommonSignals : ST_CommonSignals;
	stCommands : ST_Commands;

	// Системные переменные
	xStateEmergencyStop : BOOL := FALSE; // Флаг аварийного останова
	xStateErrorCheckReady : BOOL := FALSE; // Готовность к пуску (отсутствие ошибок)
	xStateErrorAcceptIdle : BOOL := FALSE; // Ошибка задания пропорции
	ICUR_PRECENT : REAL := 0.0; // КИУМ в процентах
	eSystemStageToSCADA : E_ScadaStatesDevice; // Общее состояние системы для SCADA

	// Шаги автоматического алгоритма
	AUTO_STEP : (
		IDLE, 				// Ожидание задания пропорции
		INIT,				// Расчёт производительности
		START_DUMPER,		// Запуск отвалообразователя
		START_CONV,			// Запуск конвейера
		START_VIBFEEDER,	// Запуск вибропитателей
		WORK,				// Работа отвалообразователя, доступ к дополнительным функциям
		END_REPORT,			// Завершение работы, формирование отчёта
		ERROR				// Состояние ошибки
		) := IDLE; // Начальное положение

	// Вспомогательные переменные
	i : INT; // Счётчик для циклов
	awModbusRegisters : ARRAY [0..99] OF WORD; // Массив Modbus регистров

	// Временные переменные для расчёта пропорций бункеров
	rWeight1, rWeight2, rWeight3 : REAL; // Индивидуальный вес каждого бункера
	rTotalWeightActive : REAL; // Суммарный вес активных бункеров

	// Начальные частоты вибропитателей (рассчитываются в INIT)
	rInitialFrequency_1 : REAL := 0.0; // Начальная частота бункера 1, Гц
	rInitialFrequency_2 : REAL := 0.0; // Начальная частота бункера 2, Гц
	rInitialFrequency_3 : REAL := 0.0; // Начальная частота бункера 3, Гц

	// Временная переменная для конвертации TIME из Modbus (секунды)
	rTempTime : REAL;

	ton_AutoTimer : TON; // Таймер автоматического режима

	nBunkerStartStep : INT := 0; // Подшаг последовательного запуска бункеров (0=бункер3, 1=задержка, 2=бункер2, 3=задержка, 4=бункер1, 5=готово)

	xAutoStopping : BOOL; // Процесс остановки
	xAutoEmergencyStopping : BOOL; // Процесс аварийной остановки
	xAutoEmergencyStoppingDependecies : BOOL; // Процесс аварийной остановки по блокировочным зависимостям
	nStopSubstage : INT := 0; // Подшаг последовательной остановки (0=бункер1, 1=задержка, 2=бункер2, 3=задержка, 4=бункер3, 5=задержка, 6=конвейер, 7=задержка, 8=отвалообразователь, 9=готово)

	// Команды автоматической аварийной остановки
	xAutoEmergencyStopBunker : ARRAY[1..3] OF BOOL; // Автоматическая аварийная остановка бункеров
	xAutoEmergencyStopConveyor : BOOL; // Автоматическая аварийная остановка конвейера
	xAutoEmergencyStopDumper : BOOL; // Автоматическая аварийная остановка отвалообразователя

	// Управление светофорами бункеров
	xCriticalWeightDetected : BOOL := FALSE; // Флаг критически низкого веса (хотя бы один бункер достиг критической уставки)
	xEmptyBunkerDetected : BOOL := FALSE; // Флаг опустошения (хотя бы один бункер полностью пуст)

	// Контроль суммы пропорций в режиме WORK
	tonProportionSumTimeout : TON; // Таймер контроля суммы пропорций
	xProportionSumError : BOOL := FALSE; // Флаг ошибки суммы пропорций (сумма не равна 100%)
	rProportionSum : REAL := 0.0; // Текущая сумма пропорций

	// Контроль минимальной и максимальной частоты вибропитателей (ПИД-регулятор)
	tonMinFrequencyTimeout : ARRAY[1..3] OF TON; // Таймеры контроля минимальной частоты для каждого бункера
	xMinFrequencyError : BOOL := FALSE; // Флаг аварии: частота вибропитателя упала ниже минимума
	tonMaxFrequencyTimeout : ARRAY[1..3] OF TON; // Таймеры контроля максимальной частоты для каждого бункера
	xMaxFrequencyError : BOOL := FALSE; // Флаг аварии: частота вибропитателя превысила максимум
END_VAR

stCommonSignals.qx6KM1 := TRUE;

// Временно
stBunker[1].rWeight := 100;
stBunker[2].rWeight := 100;
stBunker[3].rWeight := 100;

// == ИНИЦИАЛИЗАЦИЯ ==
// Инициализация общих сигналов
stCommonSignals.fbEmergencyStopBtn(
	ixSignal := , // Подключить физический вход
	xEnableRattlingFilter := FALSE // Базовый сигнал без фильтра
);

stCommonSignals.fbRemoteModeBtn(
	ixSignal := , // Подключить физический вход
	xEnableRattlingFilter := TRUE,
	tStabilityTime := T#100MS
);

stCommonSignals.fbRealyCurrentControl(
	ixSignal := , // Подключить физический вход
	xEnableRattlingFilter := TRUE,
	tStabilityTime := T#100MS
);

stCommonSignals.fbQF1(
	ixSignal := , // Подключить физический вход
	xEnableRattlingFilter := TRUE
);

stCommonSignals.fb9QF1(
	ixSignal := , // Подключить физический вход
	xEnableRattlingFilter := TRUE
);

stCommonSignals.fb10QF1(
	ixSignal := , // Подключить физический вход
	xEnableRattlingFilter := TRUE
);

stCommonSignals.fb11QF1(
	ixSignal := , // Подключить физический вход
	xEnableRattlingFilter := TRUE
);

// Инициализация команд
stCommands.cmdResetAll(
	ixSignal := , // Подключить физический вход
	xEnableRattlingFilter := FALSE // Только edge detection
);

stCommands.cmdStartCommon(
	ixSignal := , // Подключить физический вход
	xEnableRattlingFilter := FALSE // Только edge detection
);

stCommands.cmdStopCommon(
	ixSignal := , // Подключить физический вход
	xEnableRattlingFilter := FALSE // Только edge detection
);

stCommands.cmdEmergencyStopCommon(
	ixSignal := , // Подключить физический вход
	xEnableRattlingFilter := FALSE // Только edge detection
);

// == КОНТРОЛЬ СВЯЗИ СО SCADA ==
fbScadaCommunication(
	ixHeartbeatSignal := SCADA_HEARTBEAT,
	itTimeout := SCADA_HEARTBEAT_TIMEOUT,
	xReset := stCommands.cmdResetAll.qxSignal
);

// Постоянный внутренний импульс-сигнал
PULSE(ENABLE:= TRUE, TIMELOW:= T#200MS, TIMEHIGH := T#200MS);
PULSE_RTRIG(CLK:= PULSE.OUT);

// Конвертация сигнала светофора бункера в WORD
FOR i := 1 TO 3 DO
	stBunker[i].wLightColor := TO_WORD(stBunker[i].eLightColor);
END_FOR

// == ОБРАБОТКА ФУНКЦИОНАЛЬНЫХ БЛОКОВ ==
// Бункеры
fbBunker[1](
	Bunker := stBunker[1],
	xLocalMode := NOT stCommonSignals.fbRemoteModeBtn.qxSignal, // 1 - Дистанция, 0 - местный
	xStart := xStartBunker[1],
	xStop := xAutoEmergencyStopping OR xManualStopBunker[1] OR xAutoEmergencyStopBunker[1],
	xEmergencyStop := xAutoEmergencyStopBunker[1],
	xEmergencyStopVibrator := stBunker[1].cmdEmergencyStopVibrator OR xAutoEmergencyStopBunker[1],
	xReset := stCommands.cmdResetAll.qxSignal OR stBunker[1].cmdReset,
	irManualFrequency := BUNKER_1_FREQ_VIBFEEDER,
	irManualFrequencyVibrator := BUNKER_1_FREQ_VIBRATOR,
	eStage => eBunkerStage[1],
	eStageToSCADA => eBunkerStageToSCADA[1]
);

fbBunker[2](
	Bunker := stBunker[2],
	xLocalMode := NOT stCommonSignals.fbRemoteModeBtn.qxSignal, // 1 - Дистанция, 0 - местный
	xStart := xStartBunker[2],
	xStop := xAutoEmergencyStopping OR xManualStopBunker[2] OR xAutoEmergencyStopBunker[2],
	xEmergencyStop := xAutoEmergencyStopBunker[2],
	xEmergencyStopVibrator := stBunker[2].cmdEmergencyStopVibrator OR xAutoEmergencyStopBunker[2],
	xReset := stCommands.cmdResetAll.qxSignal OR stBunker[2].cmdReset,
	irManualFrequency := BUNKER_2_FREQ_VIBFEEDER,
	irManualFrequencyVibrator := BUNKER_2_FREQ_VIBRATOR,
	eStage => eBunkerStage[2],
	eStageToSCADA => eBunkerStageToSCADA[2]
);

fbBunker[3](
	Bunker := stBunker[3],
	xLocalMode := NOT stCommonSignals.fbRemoteModeBtn.qxSignal, // 1 - Дистанция, 0 - местный
	xStart := xStartBunker[3],
	xStop := xAutoEmergencyStopping OR xManualStopBunker[3] OR xAutoEmergencyStopBunker[3],
	xEmergencyStop := xAutoEmergencyStopBunker[3],
	xEmergencyStopVibrator := stBunker[3].cmdEmergencyStopVibrator OR xAutoEmergencyStopBunker[3],
	xReset := stCommands.cmdResetAll.qxSignal OR stBunker[3].cmdReset,
	irManualFrequency := BUNKER_3_FREQ_VIBFEEDER,
	irManualFrequencyVibrator := BUNKER_3_FREQ_VIBRATOR,
	eStage => eBunkerStage[3],
	eStageToSCADA => eBunkerStageToSCADA[3]
);

// Отвалообразователь
fbDumper(
	Dumper := stDumper,
	xLocalMode := NOT stCommonSignals.fbRemoteModeBtn.qxSignal, // 1 - Дистанция, 0 - местный
	xStart := xStartDumper,
	xStop := xManualStopDumper,
	xEmergencyStop := stDumper.cmdEmergencyStop OR xAutoEmergencyStopDumper,
	xReset := stCommands.cmdResetAll.qxSignal OR stDumper.cmdReset,
	eStage => eDumperStage,
	eStageToSCADA => eDumperStageToSCADA
);

// Конвейер
fbConveyor(
	Conveyor := stConveyor,
	xLocalMode := NOT stCommonSignals.fbRemoteModeBtn.qxSignal, // 1 - Дистанция, 0 - местный
	xStart := xStartConveyor,
	xStop := xManualStopConveyor,
	xEmergencyStop := stConveyor.cmdEmergencyStop OR xAutoEmergencyStopConveyor,
	xReset := stCommands.cmdResetAll.qxSignal OR stConveyor.cmdReset,
	eStage => eConveyorStage,
	eStageToSCADA => eConveyorStageToSCADA
);

// Обновление состояния Emergency Stop
xStateEmergencyStop := stCommonSignals.fbEmergencyStopBtn.qxSignal
	OR stCommands.cmdEmergencyStopCommon.qxRisingEdge;

// ========================================
// ОПРЕДЕЛЕНИЕ ОШИБКИ БЛОКИРОВОЧНЫХ ЗАВИСИМОСТЕЙ
// ========================================
// ВАЖНО: Вычисляется ДО вызова fbEmergencyStopCollector для использования в текущем цикле
//
// Блокировочные зависимости:
// 1. Бункеры работают, но конвейер или отвалообразователь НЕ в WORK
// 2. Конвейер работает, но отвалообразователь НЕ в WORK
xAutoEmergencyStoppingDependecies :=
	(NOT (eConveyorStage = E_StageWithPreStartAlarm.WORK AND eDumperStage = E_StageWithPreStartAlarm.WORK)
	AND (eBunkerStage[1] = E_StageWithPreStartAlarm.WORK
	OR eBunkerStage[2] = E_StageWithPreStartAlarm.WORK
	OR eBunkerStage[3] = E_StageWithPreStartAlarm.WORK))
	OR (eConveyorStage = E_StageWithPreStartAlarm.WORK AND NOT eDumperStage = E_StageWithPreStartAlarm.WORK);

// ========================================
// ЦЕНТРАЛИЗОВАННАЯ ОБРАБОТКА АВАРИЙНОЙ ОСТАНОВКИ
// ========================================

fbEmergencyStopCollector(
	// Гарантированные источники (NC контакты: TRUE = норма)
	ixEStopButton := stCommonSignals.fbEmergencyStopBtn.qxSignal,
	ixScadaCommand := stCommands.cmdEmergencyStopCommon.qxRisingEdge,
	ixEStopDumper := stDumper.fbBtnEmergencyStop.qxSignal,
	ixEStopConveyor := stConveyor.fbBtnEmergencyStop.qxSignal,
	ixEStopBunker1 := stBunker[1].fbBtnEmergencyStop.qxSignal,
	ixEStopBunker2 := stBunker[2].fbBtnEmergencyStop.qxSignal,
	ixEStopBunker3 := stBunker[3].fbBtnEmergencyStop.qxSignal,

	// Системные сигналы
	ixScadaLoss := fbScadaCommunication.qxCommunicationLost,
	ixProportionError := xProportionSumError,

	// Ошибки датчиков отвалообразователя (из fbDumper.fbSensors)
	ixDumperErrorZQ := fbDumper.fbSensors.xErrorZQ_Any,
	ixDumperErrorHQ := fbDumper.fbSensors.xErrorHQ_Any,
	ixDumperErrorSQ := fbDumper.fbSensors.xErrorSQ_Any,
	ixDumperErrorGS := fbDumper.fbSensors.xErrorGS,
	ixDumperErrorYS := fbDumper.fbSensors.xErrorYS,
	ixDumperErrorQR := fbDumper.fbSensors.xErrorQR_Any,

	// Ошибки датчиков конвейера (из fbConveyor.fbSensors)
	ixConveyorErrorZQ := fbConveyor.fbSensors.xErrorZQ_Any,
	ixConveyorErrorHQ := fbConveyor.fbSensors.xErrorHQ_Any,
	ixConveyorErrorSQ := fbConveyor.fbSensors.xErrorSQ_Any,
	ixConveyorErrorGS := fbConveyor.fbSensors.xErrorGS,
	ixConveyorErrorYS := fbConveyor.fbSensors.xErrorYS,
	ixConveyorErrorYE := FALSE, // Добавить когда появится металлодетектор
	ixConveyorErrorQR := fbConveyor.fbSensors.xErrorQR_Any,

	// Зависимости и ток
	ixDependencyError := xAutoEmergencyStoppingDependecies,
	ixMotorCurrentHH := FALSE, // Агрегировать из VFD при необходимости

	// Ошибки VFD (аварийный сигнал от частотного преобразователя)
	ixDumperVFD_Failure := fbDumper.fbMotorErrors.xErrorMotors,
	ixConveyorVFD_Failure := fbConveyor.fbMotorErrors.xErrorMotors,

	// Команда сброса
	ixReset := stCommands.cmdResetAll.qxRisingEdge
);

// ========================================
// СИМУЛЯЦИЯ
// ========================================

fbSimulation(
	xEnable := SIMULATION,
	xReset := ,
	Dumper := stDumper,
	Conveyor := stConveyor,
	Bunker := stBunker,
	Common := stCommonSignals
);

// == РУЧНОЙ РЕЖИМ - ДИСТАНЦИЯ ==

// ОТВАЛООБРАЗОВАТЕЛЬ

// Запуск отвалообразователя в ручном режиме
IF 	stDumper.cmdSetModeManual OR stCommands.cmdSetToManual THEN stDumper.eStateRemote := E_StateRemote.Manual; END_IF;
IF 	stDumper.cmdSetModeAuto OR stCommands.cmdSetToAuto THEN stDumper.eStateRemote := E_StateRemote.Auto; END_IF;

IF 	stDumper.eStateRemote = E_StateRemote.Manual // Находится в режиме Manual
	AND stDumper.cmdStartConveyor // Команда на запуск в ручном режиме
	AND eDumperStage <> E_StageWithPreStartAlarm.WORK // Не находится в статусе работы
	AND eDumperStage <> E_StageWithPreStartAlarm.STARTING AND eDumperStage <> E_StageWithPreStartAlarm.PRESTART_ALARM // Не в процессе запуска
	AND eDumperStage <> E_StageWithPreStartAlarm.ERROR // Не находится в ошибке
	THEN
		xManualStopDumper := FALSE;
		xStartDumper := TRUE;
END_IF;
// Сброс импульсной команды запуска после начала предпусковой сигнализации
IF (eDumperStage = E_StageWithPreStartAlarm.PRESTART_ALARM OR eDumperStage = E_StageWithPreStartAlarm.STARTING) AND xStartDumper THEN xStartDumper := FALSE; END_IF;

// Остановка отвалообразователя в ручном режиме
IF 	stDumper.eStateRemote = E_StateRemote.Manual // Находится в режиме Manual
	AND stDumper.cmdStopConveyor // Команда на остановку в ручном режиме
	AND	(eDumperStage = E_StageWithPreStartAlarm.WORK // В статусе работы
		OR eDumperStage = E_StageWithPreStartAlarm.STARTING
		OR eDumperStage = E_StageWithPreStartAlarm.PRESTART_ALARM) // В процессе запуска
	THEN
		xStartDumper := FALSE;
		xManualStopDumper := TRUE;
END_IF;
// Сброс команды остановки только после полного перехода в IDLE
IF (eDumperStage = E_StageWithPreStartAlarm.IDLE OR eDumperStage = E_StageWithPreStartAlarm.ERROR) AND xManualStopDumper THEN xManualStopDumper := FALSE; END_IF;

// СБОРНЫЙ КОНВЕЙЕР

// Запуск сборочного конвейера в ручном режиме
IF 	stConveyor.cmdSetModeManual OR stCommands.cmdSetToManual THEN stConveyor.eStateRemote := E_StateRemote.Manual; END_IF;
IF 	stConveyor.cmdSetModeAuto OR stCommands.cmdSetToAuto THEN stConveyor.eStateRemote := E_StateRemote.Auto; END_IF;

IF 	stConveyor.eStateRemote = E_StateRemote.Manual // Находится в режиме Manual
	AND stConveyor.cmdStartConveyor // Команда на запуск в ручном режиме
	AND eConveyorStage <> E_StageWithPreStartAlarm.WORK // Не находится в статусе работы
	AND eConveyorStage <> E_StageWithPreStartAlarm.STARTING AND eConveyorStage <> E_StageWithPreStartAlarm.PRESTART_ALARM // Не в процессе запуска
	AND eConveyorStage <> E_StageWithPreStartAlarm.ERROR // Не находится в ошибке
	THEN
		xStartConveyor := TRUE;
		xManualStopConveyor := FALSE;
END_IF;
// Сброс импульсной команды запуска после начала предпусковой сигнализации
IF (eConveyorStage = E_StageWithPreStartAlarm.PRESTART_ALARM OR eConveyorStage = E_StageWithPreStartAlarm.STARTING) AND xStartConveyor THEN xStartConveyor := FALSE; END_IF;

// Остановка сборочного конвейера в ручном режиме
IF 	stConveyor.eStateRemote = E_StateRemote.Manual // Находится в режиме Manual
	AND stConveyor.cmdStopConveyor // Команда на остановку в ручном режиме
	AND	(eConveyorStage = E_StageWithPreStartAlarm.WORK // В статусе работы
		OR eConveyorStage = E_StageWithPreStartAlarm.STARTING
		OR eConveyorStage = E_StageWithPreStartAlarm.PRESTART_ALARM) // В процессе запуска
	THEN
		xStartConveyor := FALSE;
		xManualStopConveyor := TRUE;
END_IF;
// Сброс команды остановки только после полного перехода в IDLE
IF (eConveyorStage = E_StageWithPreStartAlarm.IDLE OR eConveyorStage = E_StageWithPreStartAlarm.ERROR) AND xManualStopConveyor THEN xManualStopConveyor := FALSE; END_IF;

// БУНКЕР 1

// Переключение режимов
IF stBunker[1].cmdSetModeManual OR stCommands.cmdSetToManual THEN stBunker[1].eStateRemote := E_StateRemote.Manual; END_IF;
IF stBunker[1].cmdSetModeAuto OR stCommands.cmdSetToAuto THEN stBunker[1].eStateRemote := E_StateRemote.Auto; END_IF;

// Запуск бункера в ручном режиме
IF stBunker[1].eStateRemote = E_StateRemote.Manual // Находится в режиме Manual
	AND stBunker[1].cmdStartFeeder // Команда на запуск в ручном режиме
	AND eBunkerStage[1] <> E_StageWithPreStartAlarm.WORK // Не находится в статусе работы
	AND eBunkerStage[1] <> E_StageWithPreStartAlarm.STARTING AND eBunkerStage[1] <> E_StageWithPreStartAlarm.PRESTART_ALARM // Не в процессе запуска
	AND eBunkerStage[1] <> E_StageWithPreStartAlarm.ERROR // Не находится в ошибке
	THEN
		xManualStopBunker[1] := FALSE;
		xStartBunker[1] := TRUE;
END_IF;
// Сброс команды запуска только после достижения статуса WORK
IF eBunkerStage[1] = E_StageWithPreStartAlarm.WORK AND xStartBunker[1] THEN xStartBunker[1] := FALSE; END_IF;

// Остановка бункера в ручном режиме
IF stBunker[1].eStateRemote = E_StateRemote.Manual // Находится в режиме Manual
	AND stBunker[1].cmdStopFeeder // Команда на остановку в ручном режиме
	AND (eBunkerStage[1] = E_StageWithPreStartAlarm.WORK // В статусе работы
		OR eBunkerStage[1] = E_StageWithPreStartAlarm.STARTING
		OR eBunkerStage[1] = E_StageWithPreStartAlarm.PRESTART_ALARM) // В процессе запуска
	THEN
		xStartBunker[1] := FALSE;
		xManualStopBunker[1] := TRUE;
END_IF;
// Сброс команды остановки только после полного перехода в IDLE
IF (eBunkerStage[1] = E_StageWithPreStartAlarm.IDLE OR eBunkerStage[1] = E_StageWithPreStartAlarm.ERROR) AND xManualStopBunker[1] THEN xManualStopBunker[1] := FALSE; END_IF;

// БУНКЕР 2

// Переключение режимов
IF stBunker[2].cmdSetModeManual OR stCommands.cmdSetToManual THEN stBunker[2].eStateRemote := E_StateRemote.Manual; END_IF;
IF stBunker[2].cmdSetModeAuto OR stCommands.cmdSetToAuto THEN stBunker[2].eStateRemote := E_StateRemote.Auto; END_IF;

// Запуск бункера в ручном режиме
IF stBunker[2].eStateRemote = E_StateRemote.Manual // Находится в режиме Manual
	AND stBunker[2].cmdStartFeeder // Команда на запуск в ручном режиме
	AND eBunkerStage[2] <> E_StageWithPreStartAlarm.WORK // Не находится в статусе работы
	AND eBunkerStage[2] <> E_StageWithPreStartAlarm.STARTING AND eBunkerStage[2] <> E_StageWithPreStartAlarm.PRESTART_ALARM // Не в процессе запуска
	AND eBunkerStage[2] <> E_StageWithPreStartAlarm.ERROR // Не находится в ошибке
	THEN
		xManualStopBunker[2] := FALSE;
		xStartBunker[2] := TRUE;
END_IF;
// Сброс команды запуска только после достижения статуса WORK
IF eBunkerStage[2] = E_StageWithPreStartAlarm.WORK AND xStartBunker[2] THEN xStartBunker[2] := FALSE; END_IF;

// Остановка бункера в ручном режиме
IF stBunker[2].eStateRemote = E_StateRemote.Manual // Находится в режиме Manual
	AND stBunker[2].cmdStopFeeder // Команда на остановку в ручном режиме
	AND (eBunkerStage[2] = E_StageWithPreStartAlarm.WORK // В статусе работы
		OR eBunkerStage[2] = E_StageWithPreStartAlarm.STARTING
		OR eBunkerStage[2] = E_StageWithPreStartAlarm.PRESTART_ALARM) // В процессе запуска
	THEN
		xStartBunker[2] := FALSE;
		xManualStopBunker[2] := TRUE;
END_IF;
// Сброс команды остановки только после полного перехода в IDLE
IF (eBunkerStage[2] = E_StageWithPreStartAlarm.IDLE OR eBunkerStage[2] = E_StageWithPreStartAlarm.ERROR) AND xManualStopBunker[2] THEN xManualStopBunker[2] := FALSE; END_IF;

// БУНКЕР 3

// Переключение режимов
IF stBunker[3].cmdSetModeManual OR stCommands.cmdSetToManual THEN stBunker[3].eStateRemote := E_StateRemote.Manual; END_IF;
IF stBunker[3].cmdSetModeAuto OR stCommands.cmdSetToAuto THEN stBunker[3].eStateRemote := E_StateRemote.Auto; END_IF;

// Запуск бункера в ручном режиме
IF stBunker[3].eStateRemote = E_StateRemote.Manual // Находится в режиме Manual
	AND stBunker[3].cmdStartFeeder // Команда на запуск в ручном режиме
	AND eBunkerStage[3] <> E_StageWithPreStartAlarm.WORK // Не находится в статусе работы
	AND eBunkerStage[3] <> E_StageWithPreStartAlarm.STARTING AND eBunkerStage[3] <> E_StageWithPreStartAlarm.PRESTART_ALARM // Не в процессе запуска
	AND eBunkerStage[3] <> E_StageWithPreStartAlarm.ERROR // Не находится в ошибке
	THEN
		xManualStopBunker[3] := FALSE;
		xStartBunker[3] := TRUE;
END_IF;
// Сброс команды запуска только после достижения статуса WORK
IF eBunkerStage[3] = E_StageWithPreStartAlarm.WORK AND xStartBunker[3] THEN xStartBunker[3] := FALSE; END_IF;

// Остановка бункера в ручном режиме
IF stBunker[3].eStateRemote = E_StateRemote.Manual // Находится в режиме Manual
	AND stBunker[3].cmdStopFeeder // Команда на остановку в ручном режиме
	AND (eBunkerStage[3] = E_StageWithPreStartAlarm.WORK // В статусе работы
		OR eBunkerStage[3] = E_StageWithPreStartAlarm.STARTING
		OR eBunkerStage[3] = E_StageWithPreStartAlarm.PRESTART_ALARM) // В процессе запуска
	THEN
		xStartBunker[3] := FALSE;
		xManualStopBunker[3] := TRUE;
END_IF;
// Сброс команды остановки только после полного перехода в IDLE
IF (eBunkerStage[3] = E_StageWithPreStartAlarm.IDLE OR eBunkerStage[3] = E_StageWithPreStartAlarm.ERROR) AND xManualStopBunker[3] THEN xManualStopBunker[3] := FALSE; END_IF;

// Процессы аварийных остановок в ручном режиме
	// F FC_Dumper_GetErrorCommon(Dumper:=stDumper) THEN FC_Dumper_EmergencyStop(Dumper:=stDumper); END_IF;
	// F FC_Conveyor_GetErrorCommon(Conveyor:=stConveyor) THEN FC_Conveyor_EmergencyStop(Conveyor:=stConveyor); END_IF;
	//FOR i := 1 TO 3 DO
		// IF FC_Bunker_GetErrorBunker(Bunker:=stBunker[i]) THEN FC_Bunker_EmergencyStop(Bunker:=stBunker[i]); END_IF;
	//END_FOR

// == АВТОМАТИЧЕСКИЙ РЕЖИМ ==
ton_AutoTimer(PT:=T#10S);

// ========================================
// ПРОВЕРКА ГОТОВНОСТИ СИСТЕМЫ К АВТОМАТИЧЕСКОМУ ПУСКУ
// ========================================
// Готовность системы = ВСЕ условия должны быть выполнены:
// 1. Не идёт процесс остановки (xAutoStopping, xAutoEmergencyStopping)
// 2. Все секции в автоматическом режиме (Auto)
// 3. Нет зафиксированных ошибок (xStateFailure)
// 4. Секции не в стадии ERROR
// 5. Секции готовы к запуску (xSectionReady):
//    - VFD готовы к пуску (дискретный сигнал fbStateRdyToStart)
//    - Нет ошибок моторов (VFD failure)
//    - Нет ошибок по датчикам безопасности
// 6. Сумма пропорций = 100%
xStateErrorCheckReady :=
	// 1. Не идёт остановка
	NOT xAutoStopping AND NOT xAutoEmergencyStopping
	// 2. Все секции в автоматическом режиме
	AND stBunker[1].eStateRemote = E_StateRemote.Auto
	AND stBunker[2].eStateRemote = E_StateRemote.Auto
	AND stBunker[3].eStateRemote = E_StateRemote.Auto
	AND stDumper.eStateRemote = E_StateRemote.Auto
	AND stConveyor.eStateRemote = E_StateRemote.Auto
	// 3. Нет зафиксированных ошибок
	AND NOT stBunker[1].xStateFailure
	AND NOT stBunker[2].xStateFailure
	AND NOT stBunker[3].xStateFailure
	AND NOT stDumper.xStateFailure
	AND NOT stConveyor.xStateFailure
	// 4. Секции не в стадии ERROR
	AND eBunkerStage[1] <> E_StageWithPreStartAlarm.ERROR
	AND eBunkerStage[2] <> E_StageWithPreStartAlarm.ERROR
	AND eBunkerStage[3] <> E_StageWithPreStartAlarm.ERROR
	AND eDumperStage <> E_StageWithPreStartAlarm.ERROR
	AND eConveyorStage <> E_StageWithPreStartAlarm.ERROR
	// 5. Секции готовы к запуску (VFD готовы, нет ошибок моторов/сенсоров)
	AND fbDumper.xSectionReady
	AND fbConveyor.xSectionReady
	// TODO: Добавить fbBunker[i].xSectionReady когда будет реализовано
	// 6. Сумма пропорций = 100%
	AND BUNKER_WORK_PRECENT_1 + BUNKER_WORK_PRECENT_2 + BUNKER_WORK_PRECENT_3 = 100;

// ========================================
// ОБРАБОТКА ВЫХОДОВ FB_EmergencyStopCollector
// ========================================

// Глобальная аварийная остановка (из централизованного блока)
xAutoEmergencyStopping := fbEmergencyStopCollector.qxGlobalEmergencyStop;

// Сигналы остановки по секциям (из централизованного блока)
xAutoEmergencyStopDumper := fbEmergencyStopCollector.qxSectionStop_Dumper;
xAutoEmergencyStopConveyor := fbEmergencyStopCollector.qxSectionStop_Conveyor;
xAutoEmergencyStopBunker[1] := fbEmergencyStopCollector.qxSectionStop_Bunker1;
xAutoEmergencyStopBunker[2] := fbEmergencyStopCollector.qxSectionStop_Bunker2;
xAutoEmergencyStopBunker[3] := fbEmergencyStopCollector.qxSectionStop_Bunker3;

// Сброс сигналов после остановки секций
IF xAutoEmergencyStopBunker[1] AND (eBunkerStage[1] = E_StageWithPreStartAlarm.IDLE OR eBunkerStage[1] = E_StageWithPreStartAlarm.ERROR) THEN xAutoEmergencyStopBunker[1] := FALSE; END_IF;
IF xAutoEmergencyStopBunker[2] AND (eBunkerStage[2] = E_StageWithPreStartAlarm.IDLE OR eBunkerStage[2] = E_StageWithPreStartAlarm.ERROR) THEN xAutoEmergencyStopBunker[2] := FALSE; END_IF;
IF xAutoEmergencyStopBunker[3] AND (eBunkerStage[3] = E_StageWithPreStartAlarm.IDLE OR eBunkerStage[3] = E_StageWithPreStartAlarm.ERROR) THEN xAutoEmergencyStopBunker[3] := FALSE; END_IF;
IF xAutoEmergencyStopConveyor AND (eConveyorStage = E_StageWithPreStartAlarm.IDLE OR eConveyorStage = E_StageWithPreStartAlarm.ERROR) THEN xAutoEmergencyStopConveyor := FALSE; END_IF;
IF xAutoEmergencyStopDumper AND (eDumperStage = E_StageWithPreStartAlarm.IDLE OR eDumperStage = E_StageWithPreStartAlarm.ERROR) THEN xAutoEmergencyStopDumper := FALSE; END_IF;

// Обычная остановка
IF stCommands.cmdStopCommon.qxSignal AND NOT xAutoEmergencyStopping AND AUTO_STEP <> IDLE THEN
	// Сброс команд запуска
	xStartBunker[1] := FALSE;
	xStartBunker[2] := FALSE;
	xStartBunker[3] := FALSE;
	xStartConveyor := FALSE;
	xStartDumper := FALSE;

	// Установка команд остановки для оборудования в процессе запуска
	// (чтобы прервать ППЗ/запуск)
	IF AUTO_STEP = START_DUMPER THEN
		// Отвалообразователь в ППЗ или запуске - остановить его
		xManualStopDumper := TRUE;
	ELSIF AUTO_STEP = START_CONV THEN
		// Конвейер в ППЗ или запуске - остановить его и отвалообразователь
		xManualStopConveyor := TRUE;
		xManualStopDumper := TRUE;
	ELSIF AUTO_STEP = START_VIBFEEDER THEN
		// Бункеры в процессе запуска - остановить всё
		IF eBunkerStage[1] = E_StageWithPreStartAlarm.WORK THEN xManualStopBunker[1] := TRUE; END_IF;
		IF eBunkerStage[2] = E_StageWithPreStartAlarm.WORK THEN xManualStopBunker[2] := TRUE; END_IF;
		IF eBunkerStage[3] = E_StageWithPreStartAlarm.WORK THEN xManualStopBunker[3] := TRUE; END_IF;
		xManualStopConveyor := TRUE;
		xManualStopDumper := TRUE;
		nBunkerStartStep := 0; // Сброс подшага запуска бункеров
	END_IF;

	AUTO_STEP := WORK;
	xAutoStopping := TRUE;
END_IF

CASE AUTO_STEP OF

	IDLE: // Стадия ожидания задания

	// Сброс таймера и флага ошибки пропорций
	tonProportionSumTimeout.IN := FALSE;
	xProportionSumError := FALSE;

	// Сброс таймеров и флагов ошибки минимальной/максимальной частоты
	tonMinFrequencyTimeout[1].IN := FALSE;
	tonMinFrequencyTimeout[2].IN := FALSE;
	tonMinFrequencyTimeout[3].IN := FALSE;
	xMinFrequencyError := FALSE;
	tonMaxFrequencyTimeout[1].IN := FALSE;
	tonMaxFrequencyTimeout[2].IN := FALSE;
	tonMaxFrequencyTimeout[3].IN := FALSE;
	xMaxFrequencyError := FALSE;

	// Управление светофорами бункеров в режиме ожидания
	FOR i := 1 TO 3 DO
		IF stBunker[i].eStateRemoteLighter = E_StateRemote.Auto THEN
			stBunker[i].eLightColor := FC_Bunker_GetLightColor(
				irWeight := stBunker[i].rWeight,
				xCriticalWeightDetected := FALSE, // В режиме IDLE критический вес не проверяется
				xThisBunkerIsCritical := FALSE,
				xBunkerWorking := FALSE
			);

			FC_Bunker_SetLightColor(
				Bunker := stBunker[i],
				eColor := stBunker[i].eLightColor
			);
		END_IF;
	END_FOR;

	IF stCommands.cmdStartCommon.qxSignal AND xStateErrorCheckReady THEN
		AUTO_STEP := INIT;
	END_IF;

	INIT : // Первоначальный расчёт работы вибропитателей
		// Расчёт начальных частот на основе заданных пропорций
		// Формула: FreqBase_i = TargetSum * (Proportion_i / 100)

		rInitialFrequency_1 := BUNKER_VIBFEEDER_FREQUENCY_TARGET_SUM * (BUNKER_WORK_PRECENT_1 / 100.0);
		rInitialFrequency_2 := BUNKER_VIBFEEDER_FREQUENCY_TARGET_SUM * (BUNKER_WORK_PRECENT_2 / 100.0);
		rInitialFrequency_3 := BUNKER_VIBFEEDER_FREQUENCY_TARGET_SUM * (BUNKER_WORK_PRECENT_3 / 100.0);

		// ВАЖНО: Частоты НЕ записываются сразу в структуры бункеров
		// Они будут установлены индивидуально при запуске каждого бункера в START_VIBFEEDER

		// Переход к запуску отвалообразователя
		AUTO_STEP := START_DUMPER;

	START_DUMPER :
		// Запуск отвалообразователя
		// (обработка остановки перенесена в секцию "Обычная остановка" выше CASE)
		IF eDumperStage <> E_StageWithPreStartAlarm.WORK THEN
			xStartDumper := TRUE; // Команда запуска отвалообразователя
		ELSE
			xStartDumper := FALSE; // Гарантированный сброс команды при достижении WORK
			ton_AutoTimer.IN := TRUE;
			IF ton_AutoTimer.Q THEN
				ton_AutoTimer.IN := FALSE;
				AUTO_STEP := START_CONV; // Отвалообразователь запущен, переход к следующему шагу
			END_IF;
		END_IF;

	START_CONV:
		// Запуск конвейера
		// (обработка остановки перенесена в секцию "Обычная остановка" выше CASE)
		IF eConveyorStage <> E_StageWithPreStartAlarm.WORK THEN
			xStartConveyor := TRUE; // Команда запуска конвейера
		ELSE
			xStartConveyor := FALSE; // Гарантированный сброс команды при достижении WORK
			ton_AutoTimer.IN := TRUE;
			IF ton_AutoTimer.Q THEN
				ton_AutoTimer.IN := FALSE;
				AUTO_STEP := START_VIBFEEDER; // Конвейер запущен, переход к следующему шагу
			END_IF;
		END_IF;

	START_VIBFEEDER:
		// Запуск вибропитателей
		// (обработка остановки перенесена в секцию "Обычная остановка" выше CASE)

		// Последовательный запуск бункеров с задержкой: 3 → задержка → 2 → задержка → 1
		// ВАЖНО: Частота задаётся ПЕРЕД запуском каждого бункера
		CASE nBunkerStartStep OF
			0: // Шаг 0: Запуск бункера 3
				IF stBunker[3].eStateRemote = E_StateRemote.Auto AND BUNKER_WORK_PRECENT_3 > 0 THEN
					// Установка частоты ПЕРЕД запуском бункера 3
					stBunker[3].rMotorVibFeederCommonFrequency := BUNKER_3_FREQ_VIBFEEDER; // TODO ВРЕМЕННО rInitialFrequency_3
					xStartBunker[3] := TRUE;
					IF eBunkerStage[3] = E_StageWithPreStartAlarm.WORK THEN
						xStartBunker[3] := FALSE;
						nBunkerStartStep := 1; // Бункер 3 запущен → задержка
					END_IF;
				ELSE
					xStartBunker[3] := FALSE; // Гарантированный сброс при пропуске
					nBunkerStartStep := 2; // Бункер 3 пропущен → переход к бункеру 2 без задержки
				END_IF;

			1: // Шаг 1: Задержка после бункера 3
				ton_AutoTimer.IN := TRUE;
				IF ton_AutoTimer.Q THEN
					ton_AutoTimer.IN := FALSE;
					nBunkerStartStep := 2; // Переход к бункеру 2
				END_IF;

			2: // Шаг 2: Запуск бункера 2
				IF stBunker[2].eStateRemote = E_StateRemote.Auto AND BUNKER_WORK_PRECENT_2 > 0 THEN
					// Установка частоты ПЕРЕД запуском бункера 2
					stBunker[2].rMotorVibFeederCommonFrequency := BUNKER_2_FREQ_VIBFEEDER; // TODO ВРЕМЕННО rInitialFrequency_2
					xStartBunker[2] := TRUE;
					IF eBunkerStage[2] = E_StageWithPreStartAlarm.WORK THEN
						xStartBunker[2] := FALSE;
						nBunkerStartStep := 3; // Бункер 2 запущен → задержка
					END_IF;
				ELSE
					xStartBunker[2] := FALSE; // Гарантированный сброс при пропуске
					nBunkerStartStep := 4; // Бункер 2 пропущен → переход к бункеру 1 без задержки
				END_IF;

			3: // Шаг 3: Задержка после бункера 2
				ton_AutoTimer.IN := TRUE;
				IF ton_AutoTimer.Q THEN
					ton_AutoTimer.IN := FALSE;
					nBunkerStartStep := 4; // Переход к бункеру 1
				END_IF;

			4: // Шаг 4: Запуск бункера 1
				IF stBunker[1].eStateRemote = E_StateRemote.Auto AND BUNKER_WORK_PRECENT_1 > 0 THEN
					// Установка частоты ПЕРЕД запуском бункера 1
					stBunker[1].rMotorVibFeederCommonFrequency := BUNKER_1_FREQ_VIBFEEDER; // TODO ВРЕМЕННО rInitialFrequency_1
					xStartBunker[1] := TRUE;
					IF eBunkerStage[1] = E_StageWithPreStartAlarm.WORK THEN
						xStartBunker[1] := FALSE;
						nBunkerStartStep := 5; // Бункер 1 запущен → завершение
					END_IF;
				ELSE
					xStartBunker[1] := FALSE; // Гарантированный сброс при пропуске
					nBunkerStartStep := 5; // Бункер 1 пропущен → завершение
				END_IF;

			5: // Шаг 5: Все бункеры запущены
				nBunkerStartStep := 0; // Сброс для следующего цикла
				AUTO_STEP := WORK; // Переход к работе
		END_CASE;

	WORK:
		// Нормальная работа
		xStateAutoWorking := TRUE;

		// === КОНТРОЛЬ СУММЫ ПРОПОРЦИЙ ===
		// Проверка: сумма заданных пропорций должна быть равна 100%
		rProportionSum := BUNKER_WORK_PRECENT_1 + BUNKER_WORK_PRECENT_2 + BUNKER_WORK_PRECENT_3;

		// Запуск таймера, если сумма не равна 100%
		tonProportionSumTimeout(
			IN := (rProportionSum < 99.9 OR rProportionSum > 100.1), // Допуск ±0.1%
			PT := BUNKER_PROPORTION_SUM_TIMEOUT
		);

		// Установка флага ошибки при истечении таймера
		IF tonProportionSumTimeout.Q THEN
			xProportionSumError := TRUE;
		END_IF

		// Сброс флага ошибки при корректировке пропорций
		IF rProportionSum >= 99.9 AND rProportionSum <= 100.1 THEN
			xProportionSumError := FALSE;
		END_IF

		// === КОНТРОЛЬ МИНИМАЛЬНОЙ ЧАСТОТЫ ВИБРОПИТАТЕЛЕЙ ===
		// Проверка: если частота вибропитателя упала до минимума (<=), запускаем таймер
		// При истечении таймера - аварийная остановка всего комплекса

		// Бункер 1
		tonMinFrequencyTimeout[1](
			IN := (BUNKER_WORK_PRECENT_1 > 0.0 AND fbProportionPid.qrFrequency_1 <= BUNKER_VIBFEEDER_MIN_FREQUENCY_LIMIT),
			PT := BUNKER_VIBFEEDER_MIN_FREQUENCY_TIMEOUT
		);

		// Бункер 2
		tonMinFrequencyTimeout[2](
			IN := (BUNKER_WORK_PRECENT_2 > 0.0 AND fbProportionPid.qrFrequency_2 <= BUNKER_VIBFEEDER_MIN_FREQUENCY_LIMIT),
			PT := BUNKER_VIBFEEDER_MIN_FREQUENCY_TIMEOUT
		);

		// Бункер 3
		tonMinFrequencyTimeout[3](
			IN := (BUNKER_WORK_PRECENT_3 > 0.0 AND fbProportionPid.qrFrequency_3 <= BUNKER_VIBFEEDER_MIN_FREQUENCY_LIMIT),
			PT := BUNKER_VIBFEEDER_MIN_FREQUENCY_TIMEOUT
		);

		// Установка флага аварии при срабатывании ЛЮБОГО таймера
		IF tonMinFrequencyTimeout[1].Q OR tonMinFrequencyTimeout[2].Q OR tonMinFrequencyTimeout[3].Q THEN
			xMinFrequencyError := TRUE;
		END_IF

		// === КОНТРОЛЬ МАКСИМАЛЬНОЙ ЧАСТОТЫ ВИБРОПИТАТЕЛЕЙ ===
		// Проверка: если частота вибропитателя превысила максимум (>=), запускаем таймер
		// При истечении таймера - аварийная остановка всего комплекса

		// Бункер 1
		tonMaxFrequencyTimeout[1](
			IN := (BUNKER_WORK_PRECENT_1 > 0.0 AND fbProportionPid.qrFrequency_1 >= BUNKER_VIBFEEDER_MAX_FREQUENCY_LIMIT),
			PT := BUNKER_VIBFEEDER_MAX_FREQUENCY_TIMEOUT
		);

		// Бункер 2
		tonMaxFrequencyTimeout[2](
			IN := (BUNKER_WORK_PRECENT_2 > 0.0 AND fbProportionPid.qrFrequency_2 >= BUNKER_VIBFEEDER_MAX_FREQUENCY_LIMIT),
			PT := BUNKER_VIBFEEDER_MAX_FREQUENCY_TIMEOUT
		);

		// Бункер 3
		tonMaxFrequencyTimeout[3](
			IN := (BUNKER_WORK_PRECENT_3 > 0.0 AND fbProportionPid.qrFrequency_3 >= BUNKER_VIBFEEDER_MAX_FREQUENCY_LIMIT),
			PT := BUNKER_VIBFEEDER_MAX_FREQUENCY_TIMEOUT
		);

		// Установка флага аварии при срабатывании ЛЮБОГО таймера
		IF tonMaxFrequencyTimeout[1].Q OR tonMaxFrequencyTimeout[2].Q OR tonMaxFrequencyTimeout[3].Q THEN
			xMaxFrequencyError := TRUE;
		END_IF

		// === ОБЫЧНАЯ ОСТАНОВКА ===
		IF xAutoStopping THEN
			// === БЫСТРЫЙ ВЫХОД: если всё оборудование уже остановлено ===
			// Актуально когда СТОП нажат во время ППЗ - оборудование уже в IDLE
			IF eDumperStage = E_StageWithPreStartAlarm.IDLE
				AND eConveyorStage = E_StageWithPreStartAlarm.IDLE
				AND eBunkerStage[1] <> E_StageWithPreStartAlarm.WORK
				AND eBunkerStage[2] <> E_StageWithPreStartAlarm.WORK
				AND eBunkerStage[3] <> E_StageWithPreStartAlarm.WORK
			THEN
				// Всё уже остановлено - завершить процесс остановки немедленно
				ton_AutoTimer.IN := FALSE;
				xAutoStopping := FALSE;
				xStateAutoWorking := FALSE;
				xManualStopBunker[1] := FALSE;
				xManualStopBunker[2] := FALSE;
				xManualStopBunker[3] := FALSE;
				xManualStopConveyor := FALSE;
				xManualStopDumper := FALSE;
				nStopSubstage := 0;
				AUTO_STEP := IDLE;
			// Выбор режима остановки бункеров
			ELSIF BUNKER_INSTANT_STOP THEN
				// === МГНОВЕННАЯ ОСТАНОВКА ВСЕХ БУНКЕРОВ (параллельно) ===
				CASE nStopSubstage OF
					0: // Шаг 0: Одновременная остановка всех 3-х бункеров
						IF BUNKER_WORK_PRECENT_1 > 0 THEN xManualStopBunker[1] := TRUE; END_IF
						IF BUNKER_WORK_PRECENT_2 > 0 THEN xManualStopBunker[2] := TRUE; END_IF
						IF BUNKER_WORK_PRECENT_3 > 0 THEN xManualStopBunker[3] := TRUE; END_IF

						// Ожидание остановки всех активных бункеров
						IF (BUNKER_WORK_PRECENT_1 = 0 OR eBunkerStage[1] <> E_StageWithPreStartAlarm.WORK)
						AND (BUNKER_WORK_PRECENT_2 = 0 OR eBunkerStage[2] <> E_StageWithPreStartAlarm.WORK)
						AND (BUNKER_WORK_PRECENT_3 = 0 OR eBunkerStage[3] <> E_StageWithPreStartAlarm.WORK)
						THEN
							xManualStopBunker[1] := FALSE;
							xManualStopBunker[2] := FALSE;
							xManualStopBunker[3] := FALSE;
							nStopSubstage := 1; // Все бункеры остановлены → задержка
						END_IF

					1: // Шаг 1: Задержка после остановки бункеров
						ton_AutoTimer.IN := TRUE;
						IF ton_AutoTimer.Q THEN
							ton_AutoTimer.IN := FALSE;
							nStopSubstage := 6; // Переход к остановке конвейера (пропускаем шаги 2-5)
						END_IF

					6: // Шаг 6: Остановка конвейера
						xManualStopConveyor := TRUE;
						IF eConveyorStage <> E_StageWithPreStartAlarm.WORK THEN
							xManualStopConveyor := FALSE;
							nStopSubstage := 7; // Конвейер остановлен → задержка
						END_IF

					7: // Шаг 7: Задержка после конвейера
						ton_AutoTimer.IN := TRUE;
						IF ton_AutoTimer.Q THEN
							ton_AutoTimer.IN := FALSE;
							nStopSubstage := 8; // Переход к отвалообразователю
						END_IF

					8: // Шаг 8: Остановка отвалообразователя
						xManualStopDumper := TRUE;
						IF eDumperStage <> E_StageWithPreStartAlarm.WORK THEN
							xManualStopDumper := FALSE;
							nStopSubstage := 9; // Отвалообразователь остановлен → завершение
						END_IF

					9: // Шаг 9: Завершение остановки
						ton_AutoTimer.IN := FALSE;
						xAutoStopping := FALSE;
						xStateAutoWorking := FALSE;
						nStopSubstage := 0; // Сброс для следующего цикла
						AUTO_STEP := IDLE; // Возврат в IDLE
				END_CASE
			ELSE
				// === ПОСЛЕДОВАТЕЛЬНАЯ ОСТАНОВКА БУНКЕРОВ (обратная от запуска: 3→2→1) ===
				CASE nStopSubstage OF
					0: // Шаг 0: Остановка бункера 3
						IF BUNKER_WORK_PRECENT_3 > 0 THEN
							xManualStopBunker[3] := TRUE;
							IF eBunkerStage[3] <> E_StageWithPreStartAlarm.WORK THEN
								xManualStopBunker[3] := FALSE;
								nStopSubstage := 1; // Бункер 3 остановлен → задержка
							END_IF
						ELSE
							nStopSubstage := 2; // Бункер 3 не используется → переход к бункеру 2 без задержки
						END_IF

					1: // Шаг 1: Задержка после бункера 3
						ton_AutoTimer.IN := TRUE;
						IF ton_AutoTimer.Q THEN
							ton_AutoTimer.IN := FALSE;
							nStopSubstage := 2; // Переход к бункеру 2
						END_IF

					2: // Шаг 2: Остановка бункера 2
						IF BUNKER_WORK_PRECENT_2 > 0 THEN
							xManualStopBunker[2] := TRUE;
							IF eBunkerStage[2] <> E_StageWithPreStartAlarm.WORK THEN
								xManualStopBunker[2] := FALSE;
								nStopSubstage := 3; // Бункер 2 остановлен → задержка
							END_IF
						ELSE
							nStopSubstage := 4; // Бункер 2 не используется → переход к бункеру 1 без задержки
						END_IF

					3: // Шаг 3: Задержка после бункера 2
						ton_AutoTimer.IN := TRUE;
						IF ton_AutoTimer.Q THEN
							ton_AutoTimer.IN := FALSE;
							nStopSubstage := 4; // Переход к бункеру 1
						END_IF

					4: // Шаг 4: Остановка бункера 1
						IF BUNKER_WORK_PRECENT_1 > 0 THEN
							xManualStopBunker[1] := TRUE;
							IF eBunkerStage[1] <> E_StageWithPreStartAlarm.WORK THEN
								xManualStopBunker[1] := FALSE;
								nStopSubstage := 5; // Бункер 1 остановлен → задержка
							END_IF
						ELSE
							nStopSubstage := 6; // Бункер 1 не используется → переход к конвейеру без задержки
						END_IF

					5: // Шаг 5: Задержка после бункера 1
						ton_AutoTimer.IN := TRUE;
						IF ton_AutoTimer.Q THEN
							ton_AutoTimer.IN := FALSE;
							nStopSubstage := 6; // Переход к конвейеру
						END_IF

					6: // Шаг 6: Остановка конвейера
						xManualStopConveyor := TRUE;
						IF eConveyorStage <> E_StageWithPreStartAlarm.WORK THEN
							xManualStopConveyor := FALSE;
							nStopSubstage := 7; // Конвейер остановлен → задержка
						END_IF

					7: // Шаг 7: Задержка после конвейера
						ton_AutoTimer.IN := TRUE;
						IF ton_AutoTimer.Q THEN
							ton_AutoTimer.IN := FALSE;
							nStopSubstage := 8; // Переход к отвалообразователю
						END_IF

					8: // Шаг 8: Остановка отвалообразователя
						xManualStopDumper := TRUE;
						IF eDumperStage <> E_StageWithPreStartAlarm.WORK THEN
							xManualStopDumper := FALSE;
							nStopSubstage := 9; // Отвалообразователь остановлен → завершение
						END_IF

					9: // Шаг 9: Завершение остановки
						ton_AutoTimer.IN := FALSE;
						xAutoStopping := FALSE;
						xStateAutoWorking := FALSE;
						nStopSubstage := 0; // Сброс для следующего цикла
						AUTO_STEP := IDLE; // Возврат в IDLE
				END_CASE
			END_IF
		END_IF

		IF BUNKER_ENABLE_PROPORTION_MONITORING THEN

			// === Расчёт актуальных пропорций бункеров ===
			// 1. Извлечь вес каждого бункера из кумулятивных показаний
			rWeight3 := stBunker[3].rWeightUnderBunker;
			rWeight2 := stBunker[2].rWeightUnderBunker - stBunker[3].rWeightUnderBunker;
			rWeight1 := stBunker[1].rWeightUnderBunker - stBunker[2].rWeightUnderBunker;

			// 2. Зажать отрицательные значения (ошибки датчиков)
			IF rWeight1 < 0.0 THEN rWeight1 := 0.0; END_IF
			IF rWeight2 < 0.0 THEN rWeight2 := 0.0; END_IF
			IF rWeight3 < 0.0 THEN rWeight3 := 0.0; END_IF

			// 3. Суммировать вес только активных бункеров
			rTotalWeightActive := 0.0;
			IF BUNKER_WORK_PRECENT_1 > 0.0 THEN
				rTotalWeightActive := rTotalWeightActive + rWeight1;
			END_IF
			IF BUNKER_WORK_PRECENT_2 > 0.0 THEN
				rTotalWeightActive := rTotalWeightActive + rWeight2;
			END_IF
			IF BUNKER_WORK_PRECENT_3 > 0.0 THEN
				rTotalWeightActive := rTotalWeightActive + rWeight3;
			END_IF

			// 4. Рассчитать пропорции
			IF rTotalWeightActive > 0.5 THEN  // Защита от деления на ноль
				// Активные бункеры
				IF BUNKER_WORK_PRECENT_1 > 0.0 THEN
					stBunker[1].rProportionActual := rWeight1 / rTotalWeightActive;
				ELSE
					stBunker[1].rProportionActual := 0.0;
				END_IF

				IF BUNKER_WORK_PRECENT_2 > 0.0 THEN
					stBunker[2].rProportionActual := rWeight2 / rTotalWeightActive;
				ELSE
					stBunker[2].rProportionActual := 0.0;
				END_IF

				IF BUNKER_WORK_PRECENT_3 > 0.0 THEN
					stBunker[3].rProportionActual := rWeight3 / rTotalWeightActive;
				ELSE
					stBunker[3].rProportionActual := 0.0;
				END_IF
			ELSE
				// Недостаточный вес - обнулить все пропорции
				stBunker[1].rProportionActual := 0.0;
				stBunker[2].rProportionActual := 0.0;
				stBunker[3].rProportionActual := 0.0;
			END_IF;
		END_IF;

		// ========================================
		// УПРАВЛЕНИЕ СВЕТОФОРАМИ БУНКЕРОВ
		// ========================================

		// 1. Проверка критически низкого веса (хотя бы один бункер достиг уставки BUNKER_WEIGHT_LIGHT_RED_SPECIAL)
		xCriticalWeightDetected := FC_Bunker_CheckCriticalWeight(
			Bunker1 := stBunker[1],
			Bunker2 := stBunker[2],
			Bunker3 := stBunker[3]
		);

		// 2. Проверка опустошения (хотя бы один бункер полностью пуст <= BUNKER_MINIMAL_WEIGHT)
		xEmptyBunkerDetected := FC_Bunker_CheckEmptyBunker(
			Bunker1 := stBunker[1],
			Bunker2 := stBunker[2],
			Bunker3 := stBunker[3]
		);

		// 3. Определение цвета светофора для каждого бункера
		FOR i := 1 TO 3 DO
			IF stBunker[i].eStateRemoteLighter = E_StateRemote.Auto THEN
				stBunker[i].eLightColor := FC_Bunker_GetLightColor(
					irWeight := stBunker[i].rWeight,
					xCriticalWeightDetected := xCriticalWeightDetected,
					xThisBunkerIsCritical := (stBunker[i].rWeight <= BUNKER_WEIGHT_LIGHT_RED_SPECIAL), // Проверка критичности ЭТОГО бункера
					xBunkerWorking := (eBunkerStage[i] = E_StageWithPreStartAlarm.WORK)
				);

				// 4. Применение сигналов светофора
				FC_Bunker_SetLightColor(
					Bunker := stBunker[i],
					eColor := stBunker[i].eLightColor
				);
			END_IF;
		END_FOR;

		// 5. Автоматическая остановка бункеров при опустошении
		// Как только один из бункеров становится пустым, останавливаем все бункеры
		// (конвейер и отвалообразователь продолжают работу для транспортировки остатков)
		IF xEmptyBunkerDetected THEN
			// Останавливаем все активные бункеры
			FOR i := 1 TO 3 DO
				IF eBunkerStage[i] = E_StageWithPreStartAlarm.WORK THEN
					xManualStopBunker[i] := TRUE;
				END_IF;
			END_FOR;
		END_IF;

	END_REPORT:
		// Формирование отчёта
		// TODO: Добавить формирование отчёта
		IF eDumperStage = E_StageWithPreStartAlarm.IDLE
		   AND eConveyorStage = E_StageWithPreStartAlarm.IDLE
		   AND (BUNKER_WORK_PRECENT_1 = 0 OR eBunkerStage[1] = E_StageWithPreStartAlarm.IDLE)
		   AND (BUNKER_WORK_PRECENT_2 = 0 OR eBunkerStage[2] = E_StageWithPreStartAlarm.IDLE)
		   AND (BUNKER_WORK_PRECENT_3 = 0 OR eBunkerStage[3] = E_StageWithPreStartAlarm.IDLE)
		THEN
			AUTO_STEP := IDLE; // Возврат в ожидание
		END_IF;

	ERROR:

		// Сброс таймера и флага ошибки пропорций
		tonProportionSumTimeout.IN := FALSE;
		xProportionSumError := FALSE;

		// Сброс таймеров и флагов ошибки минимальной/максимальной частоты
		tonMinFrequencyTimeout[1].IN := FALSE;
		tonMinFrequencyTimeout[2].IN := FALSE;
		tonMinFrequencyTimeout[3].IN := FALSE;
		xMinFrequencyError := FALSE;
		tonMaxFrequencyTimeout[1].IN := FALSE;
		tonMaxFrequencyTimeout[2].IN := FALSE;
		tonMaxFrequencyTimeout[3].IN := FALSE;
		xMaxFrequencyError := FALSE;

		// Переход в IDLE при сбросе ошибки
		IF stCommands.cmdResetAll.qxRisingEdge THEN
			AUTO_STEP := IDLE;
		END_IF;

END_CASE;

// ========================================
// ОПРЕДЕЛЕНИЕ ОБЩЕГО СОСТОЯНИЯ СИСТЕМЫ ДЛЯ SCADA
// ========================================

// Приоритет проверки: от более критичных к менее критичным
IF AUTO_STEP = ERROR THEN
	// Ошибка без активной работы
	eSystemStageToSCADA := E_ScadaStatesDevice.ERROR;

ELSIF AUTO_STEP = WORK AND (stDumper.xStateFailure OR stConveyor.xStateFailure OR stBunker[1].xStateFailure OR stBunker[2].xStateFailure OR stBunker[3].xStateFailure) THEN
	// Система работает с аварией (хотя бы одна секция в состоянии ошибки)
	eSystemStageToSCADA := E_ScadaStatesDevice.WORK_WITH_ERROR;

ELSIF AUTO_STEP = WORK AND (stDumper.xStateWarning OR stConveyor.xStateWarning OR stBunker[1].xStateWarning OR stBunker[2].xStateWarning OR stBunker[3].xStateWarning) THEN
	// Система работает с предупреждением (хотя бы одна секция имеет предупреждение)
	eSystemStageToSCADA := E_ScadaStatesDevice.WORK_WITH_WARNING;

ELSIF AUTO_STEP = WORK THEN
	// Система работает в норме (нет ошибок и предупреждений)
	eSystemStageToSCADA := E_ScadaStatesDevice.WORK;

ELSIF (AUTO_STEP = START_DUMPER OR AUTO_STEP = START_CONV OR AUTO_STEP = START_VIBFEEDER OR AUTO_STEP = INIT) THEN
	// Система в процессе запуска (инициализация или разгон оборудования)
	eSystemStageToSCADA := E_ScadaStatesDevice.STARTING;

ELSIF AUTO_STEP = IDLE AND (stDumper.xStateWarning OR stConveyor.xStateWarning OR stBunker[1].xStateWarning OR stBunker[2].xStateWarning OR stBunker[3].xStateWarning) THEN
	// Предупреждение без активной работы
	eSystemStageToSCADA := E_ScadaStatesDevice.WARNING;

ELSIF AUTO_STEP = IDLE AND
	(stDumper.xStateFailure OR stConveyor.xStateFailure OR stBunker[1].xStateFailure OR stBunker[2].xStateFailure OR stBunker[3].xStateFailure
	OR eDumperStageToSCADA = E_ScadaStatesDevice.ERROR OR eConveyorStageToSCADA = E_ScadaStatesDevice.ERROR OR eBunkerStage[1] = E_ScadaStatesDevice.ERROR OR eBunkerStage[2] = E_ScadaStatesDevice.ERROR OR eBunkerStage[3] = E_ScadaStatesDevice.ERROR)
	THEN
	// Система неготова к запуску (есть зафиксированные ошибки или секции в состоянии ERROR)
	eSystemStageToSCADA := E_ScadaStatesDevice.NOT_READY;

ELSIF AUTO_STEP = IDLE AND NOT xStateErrorCheckReady THEN
	// Система неготова к запуску (VFD не готовы, неверные пропорции, или другие условия не выполнены)
	eSystemStageToSCADA := E_ScadaStatesDevice.NOT_READY;

ELSE
	// Система готова к запуску (IDLE, все условия готовности выполнены)
	eSystemStageToSCADA := E_ScadaStatesDevice.READY;

END_IF;

// ========================================
// АВАРИЙНАЯ ОСТАНОВКА (независимо от AUTO_STEP)
// ========================================

// Аварийная остановка срабатывает в любом состоянии AUTO_STEP
IF xAutoEmergencyStopping THEN
	// Сброс всех команд запуска (чтобы после Reset не запустилось само)
	xStartBunker[1] := FALSE;
	xStartBunker[2] := FALSE;
	xStartBunker[3] := FALSE;
	xStartConveyor := FALSE;
	xStartDumper := FALSE;
	nBunkerStartStep := 0;

	// Установка флагов аварийной остановки для всех секций
	xAutoEmergencyStopBunker[1] := TRUE;
	xAutoEmergencyStopBunker[2] := TRUE;
	xAutoEmergencyStopBunker[3] := TRUE;
	xAutoEmergencyStopConveyor := TRUE;
	xAutoEmergencyStopDumper := TRUE;

	// Ожидание остановки всего оборудования
	IF eBunkerStage[1] <> E_StageWithPreStartAlarm.WORK
	AND eBunkerStage[2] <> E_StageWithPreStartAlarm.WORK
	AND eBunkerStage[3] <> E_StageWithPreStartAlarm.WORK
	AND eConveyorStage <> E_StageWithPreStartAlarm.WORK
	AND eDumperStage <> E_StageWithPreStartAlarm.WORK
	THEN
		// Сброс всех команд аварийной остановки
		xAutoEmergencyStopBunker[1] := FALSE;
		xAutoEmergencyStopBunker[2] := FALSE;
		xAutoEmergencyStopBunker[3] := FALSE;
		xAutoEmergencyStopConveyor := FALSE;
		xAutoEmergencyStopDumper := FALSE;
		xAutoEmergencyStopping := FALSE;
		nStopSubstage := 0;
		xStateAutoWorking := FALSE;
		ton_AutoTimer.IN := FALSE;
		xAutoStopping := FALSE;
		AUTO_STEP := ERROR;
	END_IF
END_IF

IF BUNKER_ENABLE_PID THEN
	// ========================================
	// ТАЙМЕР ДЛЯ ПЕРИОДИЧЕСКОГО ВЫЗОВА ПИД
	// ========================================
	// Генерация импульса каждые 500 мс для вызова ПИД-регулятора
	// Это снижает частоту обновления и делает регулирование более плавным

	tonPidTimer(
		IN := NOT xPidTimerPulse AND (AUTO_STEP = WORK) AND NOT xAutoStopping AND NOT xAutoEmergencyStopping,
		PT := T#500MS
	);

	// Генерация импульса при завершении таймера
	IF tonPidTimer.Q THEN
		xPidTimerPulse := TRUE;
	ELSE
		xPidTimerPulse := FALSE;
	END_IF

	// Детекция переднего фронта импульса
	rtPidPulse(CLK := xPidTimerPulse);

	// ========================================
	// ВЫЗОВ ПИД-РЕГУЛЯТОРА ПО ИМПУЛЬСУ
	// ========================================
	// ПИД вызывается только при переднем фронте импульса (каждые 500 мс)
	// ВАЖНО: ПИД отключается при любой остановке (обычной или аварийной)
	IF rtPidPulse.Q OR AUTO_STEP <> WORK THEN
		fbProportionPid(
			xEnable:= (AUTO_STEP = WORK) AND NOT xAutoStopping AND NOT xAutoEmergencyStopping,
			xReset:= stCommands.cmdResetAll.qxRisingEdge,

			rProportionTarget_1:= BUNKER_WORK_PRECENT_1 / 100.0,
			rProportionTarget_2:= BUNKER_WORK_PRECENT_2 / 100.0,
			rProportionTarget_3:= BUNKER_WORK_PRECENT_3 / 100.0,

			rProportionActual_1:= stBunker[1].rProportionActual,
			rProportionActual_2:= stBunker[2].rProportionActual,
			rProportionActual_3:= stBunker[3].rProportionActual,

			// Параметры ПИД-регулятора (настройка реакции на ошибку)
			rPID_Kp:= 0.4,                    // Пропорциональный коэффициент (снижен с 1.0)
			rPID_Ki:= 0.15,                   // Интегральный коэффициент (снижен с 0.2)
			rPID_Kd:= 0.01,                   // Дифференциальный коэффициент (снижен с 0.05)
			rPID_IntegralLimit:= 10.0,        // Ограничение интеграла (anti-windup)
			rPID_DerivativeFilter:= 0.8,      // Фильтр производной (увеличен с 0.1 для подавления шума)

			rFrequencyBase_1:= rInitialFrequency_1,
			rFrequencyBase_2:= rInitialFrequency_2,
			rFrequencyBase_3:= rInitialFrequency_3,

			rFrequency_Min:= BUNKER_VIBFEEDER_MIN_FREQUENCY_LIMIT,  // Минимальная частота из уставки
			rFrequency_Max:= BUNKER_VIBFEEDER_MAX_FREQUENCY_LIMIT,  // Максимальная частота из уставки
			rFrequency_TargetSum:= BUNKER_VIBFEEDER_FREQUENCY_TARGET_SUM,
			rDeltaTime:= 0.5                  // Период вызова ПИД-регулятора, сек
		);
	END_IF

	// ========================================
	// ПЕРЕДАЧА ЧАСТОТЫ ПИД РЕГУЛЯТОРА
	// ========================================
	// ВАЖНО: Частота передается ТОЛЬКО в стадии WORK
	// В других стадиях (INIT, START_VIBFEEDER) частота устанавливается вручную
	IF AUTO_STEP = WORK THEN
		stBunker[1].rMotorVibFeederCommonFrequency := fbProportionPID.qrFrequency_1;
		stBunker[2].rMotorVibFeederCommonFrequency := fbProportionPID.qrFrequency_2;
		stBunker[3].rMotorVibFeederCommonFrequency := fbProportionPID.qrFrequency_3;
	END_IF

END_IF;

// ========================================
// MODBUS РЕГИСТРЫ
// ========================================

fbModbusToSCADA(
	stBunker := stBunker,
	stDumper := stDumper,
	stConveyor := stConveyor,
	stCommonSignals := stCommonSignals,
	stCommands := stCommands,
	eBunkerStageToSCADA := eBunkerStageToSCADA,
	eConveyorStageToSCADA := eConveyorStageToSCADA,
	eDumperStageToSCADA := eDumperStageToSCADA,
	eSystemStageToSCADA := eSystemStageToSCADA,
	fbScadaCommunication := fbScadaCommunication
);

END_PROGRAM
